LIN {X 0,Y 232.971,Z 461.148,A -85,B 0,C 180,E1 -19706.542,E2 -19706.542} C_VEL
LIN {X 0,Y 232.837,Z 461.984,A -85,B 0,C 180,E1 -19710.001,E2 -19710.001} C_VEL
LIN {X 0,Y 232.861,Z 461.79,A -85,B 0,C 180,E1 -19711.73,E2 -19711.73} C_VEL
LIN {X 0,Y 232.964,Z 461.204,A -85,B 0,C 180,E1 -19713.46,E2 -19713.46} C_VEL
LIN {X 0,Y 233.433,Z 458.881,A -85,B 0,C 180,E1 -19716.917,E2 -19716.917} C_VEL
LIN {X 0,Y 234.07,Z 456.015,A -85,B 0,C 180,E1 -19719.506,E2 -19719.506} C_VEL
LIN {X 0,Y 235.043,Z 452.127,A -85,B 0,C 180,E1 -19722.082,E2 -19722.082} C_VEL
LIN {X 0,Y 236.444,Z 447.107,A -85,B 0,C 180,E1 -19724.635,E2 -19724.635} C_VEL
LIN {X 0,Y 238.156,Z 440.785,A -85,B 0,C 180,E1 -19727.164,E2 -19727.164} C_VEL
LIN {X 0,Y 240.375,Z 432.868,A -85,B 0,C 180,E1 -19729.648,E2 -19729.648} C_VEL
LIN {X 0,Y 242.397,Z 424.824,A -85,B 0,C 180,E1 -19731.689,E2 -19731.689} C_VEL
LIN {X 0,Y 244.588,Z 414.953,A -85,B 0,C 180,E1 -19733.721,E2 -19733.721} C_VEL
LIN {X 0,Y 246.59,Z 405.255,A -85,B 0,C 180,E1 -19735.31,E2 -19735.31} C_VEL
LIN {X 0,Y 245.528,Z 395.502,A -85,B 0,C 180,E1 -19736.937,E2 -19736.937} C_VEL
LIN {X 0,Y 243.4,Z 384.419,A -85,B 0,C 180,E1 -19738.585,E2 -19738.585} C_VEL
LIN {X 0,Y 240.222,Z 372.784,A -85,B 0,C 180,E1 -19740.129,E2 -19740.129} C_VEL
LIN {X 0,Y 236.054,Z 361.103,A -85,B 0,C 180,E1 -19741.536,E2 -19741.536} C_VEL
LIN {X 0,Y 234.99,Z 358.228,A -85,B 0,C 180,E1 -19741.853,E2 -19741.853} C_VEL
LIN {X 0,Y 234.929,Z 357.743,A -85,B 0,C 180,E1 -19741.928,E2 -19741.928} C_VEL
LIN {X 0,Y 235.264,Z 354.456,A -85,B 0,C 180,E1 -19746.238,E2 -19746.238} C_VEL
LIN {X 0,Y 235.192,Z 352.491,A -85,B 0,C 180,E1 -19749.019,E2 -19749.019} C_VEL
LIN {X 0,Y 234.976,Z 350.772,A -85,B 0,C 180,E1 -19751.605,E2 -19751.605} C_VEL
LIN {X 0,Y 234.883,Z 350.23,A -85,B 0,C 180,E1 -19754.101,E2 -19754.101} C_VEL
LIN {X 0,Y 234.85,Z 350.231,A -85,B 0,C 180,E1 -19758.825,E2 -19758.825} C_VEL
LIN {X 0,Y 234.918,Z 350.222,A -85,B 0,C 180,E1 -19761.078,E2 -19761.078} C_VEL
LIN {X 0,Y 234.923,Z 350.221,A -85,B 0,C 180,E1 -19765.36,E2 -19765.36} C_VEL
LIN {X 0,Y 234.898,Z 350.226,A -85,B 0,C 180,E1 -19769.427,E2 -19769.427} C_VEL
LIN {X 0,Y 234.968,Z 350.214,A -85,B 0,C 180,E1 -19773.806,E2 -19773.806} C_VEL
LIN {X 0,Y 234.997,Z 350.214,A -85,B 0,C 180,E1 -19778.968,E2 -19778.968} C_VEL
LIN {X 0,Y 235.096,Z 350.201,A -85,B 0,C 180,E1 -19783.059,E2 -19783.059} C_VEL
LIN {X 0,Y 235.118,Z 350.195,A -85,B 0,C 180,E1 -19787.922,E2 -19787.922} C_VEL
LIN {X 0,Y 235.376,Z 350.164,A -85,B 0,C 180,E1 -19791.414,E2 -19791.414} C_VEL
LIN {X 0,Y 235.403,Z 350.16,A -85,B 0,C 180,E1 -19793.141,E2 -19793.141} C_VEL
LIN {X 0,Y 235.592,Z 350.139,A -85,B 0,C 180,E1 -19798.29,E2 -19798.29} C_VEL
LIN {X 0,Y 235.592,Z 350.137,A -85,B 0,C 180,E1 -19801.709,E2 -19801.709} C_VEL
LIN {X 0,Y 235.372,Z 350.166,A -85,B 0,C 180,E1 -19806.86,E2 -19806.86} C_VEL
LIN {X 0,Y 235.214,Z 350.187,A -85,B 0,C 180,E1 -19810.328,E2 -19810.328} C_VEL
LIN {X 0,Y 235.111,Z 350.201,A -85,B 0,C 180,E1 -19815.607,E2 -19815.607} C_VEL
LIN {X 0,Y 235.007,Z 350.213,A -85,B 0,C 180,E1 -19819.206,E2 -19819.206} C_VEL
LIN {X 0,Y 234.946,Z 350.219,A -85,B 0,C 180,E1 -19822.884,E2 -19822.884} C_VEL
LIN {X 0,Y 234.944,Z 350.219,A -85,B 0,C 180,E1 -19826.66,E2 -19826.66} C_VEL
LIN {X 0,Y 234.898,Z 350.227,A -85,B 0,C 180,E1 -19830.573,E2 -19830.573} C_VEL
LIN {X 0,Y 234.925,Z 350.225,A -85,B 0,C 180,E1 -19834.639,E2 -19834.639} C_VEL
LIN {X 0,Y 234.922,Z 350.234,A -85,B 0,C 180,E1 -19837.287,E2 -19837.287} C_VEL
LIN {X 0,Y 235.478,Z 353.686,A -85,B 0,C 180,E1 -19841.743,E2 -19841.743} C_VEL
LIN {X 0,Y 236.045,Z 356.925,A -85,B 0,C 180,E1 -19845.609,E2 -19845.609} C_VEL
LIN {X 0,Y 236.625,Z 360.143,A -85,B 0,C 180,E1 -19849.2,E2 -19849.2} C_VEL
LIN {X 0,Y 236.789,Z 361.71,A -85,B 0,C 180,E1 -19850.867,E2 -19850.867} C_VEL
LIN {X 0,Y 236.131,Z 362.697,A -85,B 0,C 180,E1 -19851.78,E2 -19851.78} C_VEL
LIN {X 0,Y 233.267,Z 364.499,A -85,B 0,C 180,E1 -19853.194,E2 -19853.194} C_VEL
LIN {X 0,Y 230.302,Z 366.325,A -85,B 0,C 180,E1 -19854.639,E2 -19854.639} C_VEL
LIN {X 0,Y 229.536,Z 367.356,A -85,B 0,C 180,E1 -19855.588,E2 -19855.588} C_VEL
LIN {X 0,Y 229.138,Z 369.003,A -85,B 0,C 180,E1 -19857.205,E2 -19857.205} C_VEL
LIN {X 0,Y 230.068,Z 372.388,A -85,B 0,C 180,E1 -19857.554,E2 -19857.554} C_VEL
LIN {X 0,Y 233.694,Z 385.256,A -85,B 0,C 180,E1 -19858.994,E2 -19858.994} C_VEL
LIN {X 0,Y 236.083,Z 397.637,A -85,B 0,C 180,E1 -19860.546,E2 -19860.546} C_VEL
LIN {X 0,Y 237.455,Z 409.332,A -85,B 0,C 180,E1 -19862.24,E2 -19862.24} C_VEL
LIN {X 0,Y 237.876,Z 420.833,A -85,B 0,C 180,E1 -19864.164,E2 -19864.164} C_VEL
LIN {X 0,Y 237.723,Z 425.768,A -85,B 0,C 180,E1 -19865.084,E2 -19865.084} C_VEL
LIN {X 0,Y 235.114,Z 436.231,A -85,B 0,C 180,E1 -19867.133,E2 -19867.133} C_VEL
LIN {X 0,Y 232.717,Z 445.972,A -85,B 0,C 180,E1 -19869.607,E2 -19869.607} C_VEL
LIN {X 0,Y 230.397,Z 454.218,A -85,B 0,C 180,E1 -19872.239,E2 -19872.239} C_VEL
LIN {X 0,Y 228.61,Z 460.648,A -85,B 0,C 180,E1 -19874.852,E2 -19874.852} C_VEL
LIN {X 0,Y 227.307,Z 465.76,A -85,B 0,C 180,E1 -19877.5,E2 -19877.5} C_VEL
LIN {X 0,Y 226.434,Z 469.734,A -85,B 0,C 180,E1 -19880.17,E2 -19880.17} C_VEL
LIN {X 0,Y 225.853,Z 472.672,A -85,B 0,C 180,E1 -19882.849,E2 -19882.849} C_VEL
LIN {X 0,Y 225.66,Z 474.484,A -85,B 0,C 180,E1 -19885.286,E2 -19885.286} C_VEL
LIN {X 0,Y 225.663,Z 475.686,A -85,B 0,C 180,E1 -19888.215,E2 -19888.215} C_VEL
LIN {X 0,Y 225.698,Z 475.901,A -85,B 0,C 180,E1 -19889.999,E2 -19889.999} C_VEL
LIN {X 0,Y 225.662,Z 475.678,A -85,B 0,C 180,E1 -19891.784,E2 -19891.784} C_VEL
LIN {X 0,Y 225.69,Z 474.056,A -85,B 0,C 180,E1 -19895.36,E2 -19895.36} C_VEL
LIN {X 0,Y 225.852,Z 472.648,A -85,B 0,C 180,E1 -19897.149,E2 -19897.149} C_VEL
LIN {X 0,Y 226.432,Z 469.698,A -85,B 0,C 180,E1 -19899.828,E2 -19899.828} C_VEL
LIN {X 0,Y 227.306,Z 465.709,A -85,B 0,C 180,E1 -19902.498,E2 -19902.498} C_VEL
LIN {X 0,Y 228.896,Z 459.582,A -85,B 0,C 180,E1 -19905.583,E2 -19905.583} C_VEL
LIN {X 0,Y 230.724,Z 452.894,A -85,B 0,C 180,E1 -19908.192,E2 -19908.192} C_VEL
LIN {X 0,Y 232.845,Z 444.953,A -85,B 0,C 180,E1 -19910.661,E2 -19910.661} C_VEL
LIN {X 0,Y 235.088,Z 436.095,A -85,B 0,C 180,E1 -19912.868,E2 -19912.868} C_VEL
LIN {X 0,Y 237.677,Z 425.596,A -85,B 0,C 180,E1 -19914.92,E2 -19914.92} C_VEL
LIN {X 0,Y 237.746,Z 415.806,A -85,B 0,C 180,E1 -19916.683,E2 -19916.683} C_VEL
LIN {X 0,Y 237.068,Z 405.419,A -85,B 0,C 180,E1 -19918.314,E2 -19918.314} C_VEL
LIN {X 0,Y 235.7,Z 395.253,A -85,B 0,C 180,E1 -19919.722,E2 -19919.722} C_VEL
LIN {X 0,Y 232.854,Z 382.031,A -85,B 0,C 180,E1 -19921.351,E2 -19921.351} C_VEL
LIN {X 0,Y 229.624,Z 371.42,A -85,B 0,C 180,E1 -19922.526,E2 -19922.526} C_VEL
LIN {X 0,Y 229.118,Z 368.985,A -85,B 0,C 180,E1 -19922.773,E2 -19922.773} C_VEL
LIN {X 0,Y 229.704,Z 366.183,A -85,B 0,C 180,E1 -19925.542,E2 -19925.542} C_VEL
LIN {X 0,Y 229.844,Z 363.042,A -85,B 0,C 180,E1 -19928.815,E2 -19928.815} C_VEL
LIN {X 0,Y 229.425,Z 359.571,A -85,B 0,C 180,E1 -19932.676,E2 -19932.676} C_VEL
LIN {X 0,Y 228.591,Z 355.533,A -85,B 0,C 180,E1 -19937.549,E2 -19937.549} C_VEL
LIN {X 0,Y 228.078,Z 352.174,A -85,B 0,C 180,E1 -19941.955,E2 -19941.955} C_VEL
LIN {X 0,Y 227.867,Z 351.102,A -85,B 0,C 180,E1 -19943.713,E2 -19943.713} C_VEL
LIN {X 0,Y 227.873,Z 351.102,A -85,B 0,C 180,E1 -19946.377,E2 -19946.377} C_VEL
LIN {X 0,Y 227.87,Z 351.104,A -85,B 0,C 180,E1 -19950.431,E2 -19950.431} C_VEL
LIN {X 0,Y 227.896,Z 351.099,A -85,B 0,C 180,E1 -19954.422,E2 -19954.422} C_VEL
LIN {X 0,Y 227.949,Z 351.091,A -85,B 0,C 180,E1 -19958.286,E2 -19958.286} C_VEL
LIN {X 0,Y 228.028,Z 351.081,A -85,B 0,C 180,E1 -19962.826,E2 -19962.826} C_VEL
LIN {X 0,Y 228.086,Z 351.073,A -85,B 0,C 180,E1 -19967.544,E2 -19967.544} C_VEL
LIN {X 0,Y 228.3,Z 351.046,A -85,B 0,C 180,E1 -19971.146,E2 -19971.146} C_VEL
LIN {X 0,Y 228.349,Z 351.04,A -85,B 0,C 180,E1 -19972.928,E2 -19972.928} C_VEL
LIN {X 0,Y 228.547,Z 351.016,A -85,B 0,C 180,E1 -19978.238,E2 -19978.238} C_VEL
LIN {X 0,Y 228.546,Z 351.016,A -85,B 0,C 180,E1 -19981.762,E2 -19981.762} C_VEL
LIN {X 0,Y 228.351,Z 351.041,A -85,B 0,C 180,E1 -19987.072,E2 -19987.072} C_VEL
LIN {X 0,Y 228.161,Z 351.063,A -85,B 0,C 180,E1 -19990.651,E2 -19990.651} C_VEL
LIN {X 0,Y 228.058,Z 351.074,A -85,B 0,C 180,E1 -19994.273,E2 -19994.273} C_VEL
LIN {X 0,Y 227.997,Z 351.084,A -85,B 0,C 180,E1 -19997.954,E2 -19997.954} C_VEL
LIN {X 0,Y 227.916,Z 351.092,A -85,B 0,C 180,E1 -20002.325,E2 -20002.325} C_VEL
LIN {X 0,Y 227.916,Z 351.095,A -85,B 0,C 180,E1 -20006.593,E2 -20006.593} C_VEL
LIN {X 0,Y 227.868,Z 351.101,A -85,B 0,C 180,E1 -20010.281,E2 -20010.281} C_VEL
LIN {X 0,Y 227.872,Z 351.1,A -85,B 0,C 180,E1 -20013.722,E2 -20013.722} C_VEL
LIN {X 0,Y 227.839,Z 351.104,A -85,B 0,C 180,E1 -20018.092,E2 -20018.092} C_VEL
LIN {X 0,Y 227.789,Z 351.111,A -85,B 0,C 180,E1 -20022.748,E2 -20022.748} C_VEL
LIN {X 0,Y 227.855,Z 351.213,A -85,B 0,C 180,E1 -20027.27,E2 -20027.27} C_VEL
LIN {X 0,Y 228.109,Z 353.189,A -85,B 0,C 180,E1 -20030.376,E2 -20030.376} C_VEL
LIN {X 0,Y 228.239,Z 355.821,A -85,B 0,C 180,E1 -20034.195,E2 -20034.195} C_VEL
LIN {X 0,Y 228.018,Z 357.999,A -85,B 0,C 180,E1 -20037.156,E2 -20037.156} C_VEL
LIN {X 0,Y 229.088,Z 361.247,A -85,B 0,C 180,E1 -20037.526,E2 -20037.526} C_VEL
LIN {X 0,Y 233.181,Z 372.217,A -85,B 0,C 180,E1 -20038.935,E2 -20038.935} C_VEL
LIN {X 0,Y 236.434,Z 383.735,A -85,B 0,C 180,E1 -20040.529,E2 -20040.529} C_VEL
LIN {X 0,Y 238.509,Z 394.227,A -85,B 0,C 180,E1 -20042.128,E2 -20042.128} C_VEL
LIN {X 0,Y 239.672,Z 403.1,A -85,B 0,C 180,E1 -20043.639,E2 -20043.639} C_VEL
LIN {X 0,Y 239.797,Z 407.32,A -85,B 0,C 180,E1 -20044.388,E2 -20044.388} C_VEL
LIN {X 0,Y 237.437,Z 417.763,A -85,B 0,C 180,E1 -20046.218,E2 -20046.218} C_VEL
LIN {X 0,Y 235.421,Z 426.646,A -85,B 0,C 180,E1 -20048.185,E2 -20048.185} C_VEL
LIN {X 0,Y 232.983,Z 435.524,A -85,B 0,C 180,E1 -20050.622,E2 -20050.622} C_VEL
LIN {X 0,Y 230.792,Z 442.926,A -85,B 0,C 180,E1 -20053.186,E2 -20053.186} C_VEL
LIN {X 0,Y 229.094,Z 448.862,A -85,B 0,C 180,E1 -20055.794,E2 -20055.794} C_VEL
LIN {X 0,Y 227.744,Z 453.551,A -85,B 0,C 180,E1 -20058.43,E2 -20058.43} C_VEL
LIN {X 0,Y 226.795,Z 457.137,A -85,B 0,C 180,E1 -20061.088,E2 -20061.088} C_VEL
LIN {X 0,Y 226.238,Z 459.716,A -85,B 0,C 180,E1 -20063.76,E2 -20063.76} C_VEL
LIN {X 0,Y 225.881,Z 461.364,A -85,B 0,C 180,E1 -20066.433,E2 -20066.433} C_VEL
LIN {X 0,Y 225.778,Z 461.971,A -85,B 0,C 180,E1 -20068.217,E2 -20068.217} C_VEL
LIN {X 0,Y 225.751,Z 462.199,A -85,B 0,C 180,E1 -20070.001,E2 -20070.001} C_VEL
LIN {X 0,Y 225.778,Z 462.005,A -85,B 0,C 180,E1 -20071.785,E2 -20071.785} C_VEL
LIN {X 0,Y 226.06,Z 460.453,A -85,B 0,C 180,E1 -20075.352,E2 -20075.352} C_VEL
LIN {X 0,Y 226.394,Z 459.096,A -85,B 0,C 180,E1 -20077.134,E2 -20077.134} C_VEL
LIN {X 0,Y 227.07,Z 456.23,A -85,B 0,C 180,E1 -20079.802,E2 -20079.802} C_VEL
LIN {X 0,Y 228.109,Z 452.341,A -85,B 0,C 180,E1 -20082.455,E2 -20082.455} C_VEL
LIN {X 0,Y 229.581,Z 447.321,A -85,B 0,C 180,E1 -20085.083,E2 -20085.083} C_VEL
LIN {X 0,Y 231.38,Z 440.998,A -85,B 0,C 180,E1 -20087.683,E2 -20087.683} C_VEL
LIN {X 0,Y 233.706,Z 433.08,A -85,B 0,C 180,E1 -20090.233,E2 -20090.233} C_VEL
LIN {X 0,Y 235.703,Z 425.511,A -85,B 0,C 180,E1 -20092.214,E2 -20092.214} C_VEL
LIN {X 0,Y 237.845,Z 416.231,A -85,B 0,C 180,E1 -20094.204,E2 -20094.204} C_VEL
LIN {X 0,Y 239.95,Z 406.756,A -85,B 0,C 180,E1 -20095.829,E2 -20095.829} C_VEL
LIN {X 0,Y 239.062,Z 397.402,A -85,B 0,C 180,E1 -20097.473,E2 -20097.473} C_VEL
LIN {X 0,Y 237.101,Z 386.551,A -85,B 0,C 180,E1 -20099.192,E2 -20099.192} C_VEL
LIN {X 0,Y 234.225,Z 375.555,A -85,B 0,C 180,E1 -20100.763,E2 -20100.763} C_VEL
LIN {X 0,Y 230.277,Z 364.192,A -85,B 0,C 180,E1 -20102.255,E2 -20102.255} C_VEL
LIN {X 0,Y 228.124,Z 358.66,A -85,B 0,C 180,E1 -20102.921,E2 -20102.921} C_VEL
LIN {X 0,Y 228.02,Z 357.983,A -85,B 0,C 180,E1 -20103.015,E2 -20103.015} C_VEL
LIN {X 0,Y 228.248,Z 355.211,A -85,B 0,C 180,E1 -20106.815,E2 -20106.815} C_VEL
LIN {X 0,Y 228.052,Z 352.842,A -85,B 0,C 180,E1 -20110.329,E2 -20110.329} C_VEL
LIN {X 0,Y 227.856,Z 351.327,A -85,B 0,C 180,E1 -20112.732,E2 -20112.732} C_VEL
LIN {X 0,Y 227.821,Z 351.11,A -85,B 0,C 180,E1 -20115.196,E2 -20115.196} C_VEL
LIN {X 0,Y 227.798,Z 351.111,A -85,B 0,C 180,E1 -20119.617,E2 -20119.617} C_VEL
LIN {X 0,Y 227.864,Z 351.101,A -85,B 0,C 180,E1 -20124.125,E2 -20124.125} C_VEL
LIN {X 0,Y 227.856,Z 351.099,A -85,B 0,C 180,E1 -20128.375,E2 -20128.375} C_VEL
LIN {X 0,Y 227.854,Z 351.101,A -85,B 0,C 180,E1 -20132.441,E2 -20132.441} C_VEL
LIN {X 0,Y 227.894,Z 351.096,A -85,B 0,C 180,E1 -20136.365,E2 -20136.365} C_VEL
LIN {X 0,Y 227.937,Z 351.091,A -85,B 0,C 180,E1 -20140.174,E2 -20140.174} C_VEL
LIN {X 0,Y 228.057,Z 351.076,A -85,B 0,C 180,E1 -20143.898,E2 -20143.898} C_VEL
LIN {X 0,Y 228.074,Z 351.073,A -85,B 0,C 180,E1 -20147.543,E2 -20147.543} C_VEL
LIN {X 0,Y 228.306,Z 351.046,A -85,B 0,C 180,E1 -20151.146,E2 -20151.146} C_VEL
LIN {X 0,Y 228.354,Z 351.039,A -85,B 0,C 180,E1 -20152.928,E2 -20152.928} C_VEL
LIN {X 0,Y 228.551,Z 351.016,A -85,B 0,C 180,E1 -20158.238,E2 -20158.238} C_VEL
LIN {X 0,Y 228.551,Z 351.014,A -85,B 0,C 180,E1 -20161.762,E2 -20161.762} C_VEL
LIN {X 0,Y 228.323,Z 351.044,A -85,B 0,C 180,E1 -20167.072,E2 -20167.072} C_VEL
LIN {X 0,Y 228.145,Z 351.066,A -85,B 0,C 180,E1 -20170.651,E2 -20170.651} C_VEL
LIN {X 0,Y 228.062,Z 351.08,A -85,B 0,C 180,E1 -20174.272,E2 -20174.272} C_VEL
LIN {X 0,Y 228.002,Z 351.086,A -85,B 0,C 180,E1 -20177.953,E2 -20177.953} C_VEL
LIN {X 0,Y 227.921,Z 351.094,A -85,B 0,C 180,E1 -20182.324,E2 -20182.324} C_VEL
LIN {X 0,Y 227.922,Z 351.094,A -85,B 0,C 180,E1 -20186.592,E2 -20186.592} C_VEL
LIN {X 0,Y 227.873,Z 351.102,A -85,B 0,C 180,E1 -20190.281,E2 -20190.281} C_VEL
LIN {X 0,Y 227.876,Z 351.103,A -85,B 0,C 180,E1 -20193.721,E2 -20193.721} C_VEL
LIN {X 0,Y 227.916,Z 351.27,A -85,B 0,C 180,E1 -20196.704,E2 -20196.704} C_VEL
LIN {X 0,Y 228.32,Z 353.894,A -85,B 0,C 180,E1 -20200.272,E2 -20200.272} C_VEL
LIN {X 0,Y 228.979,Z 357.739,A -85,B 0,C 180,E1 -20205.095,E2 -20205.095} C_VEL
LIN {X 0,Y 229.569,Z 360.957,A -85,B 0,C 180,E1 -20208.839,E2 -20208.839} C_VEL
LIN {X 0,Y 229.799,Z 364.142,A -85,B 0,C 180,E1 -20212.29,E2 -20212.29} C_VEL
LIN {X 0,Y 229.536,Z 367.356,A -85,B 0,C 180,E1 -20215.588,E2 -20215.588} C_VEL
LIN {X 0,Y 229.594,Z 369.045,A -85,B 0,C 180,E1 -20216.42,E2 -20216.42} C_VEL
LIN {X 0,Y 229.811,Z 371.78,A -85,B 0,C 180,E1 -20217.075,E2 -20217.075} C_VEL
LIN {X 0,Y 230.043,Z 376.979,A -85,B 0,C 180,E1 -20217.779,E2 -20217.779} C_VEL
LIN {X 0,Y 229.617,Z 387.244,A -85,B 0,C 180,E1 -20218.563,E2 -20218.563} C_VEL
LIN {X 0,Y 228.964,Z 393.373,A -85,B 0,C 180,E1 -20219.082,E2 -20219.082} C_VEL
LIN {X 0,Y 229.078,Z 395.306,A -85,B 0,C 180,E1 -20219.316,E2 -20219.316} C_VEL
LIN {X 0,Y 230.658,Z 407.037,A -85,B 0,C 180,E1 -20221.043,E2 -20221.043} C_VEL
LIN {X 0,Y 231.246,Z 417.991,A -85,B 0,C 180,E1 -20222.878,E2 -20222.878} C_VEL
LIN {X 0,Y 230.995,Z 426.732,A -85,B 0,C 180,E1 -20224.548,E2 -20224.548} C_VEL
LIN {X 0,Y 228.568,Z 436.018,A -85,B 0,C 180,E1 -20226.439,E2 -20226.439} C_VEL
LIN {X 0,Y 226.272,Z 444.877,A -85,B 0,C 180,E1 -20228.717,E2 -20228.717} C_VEL
LIN {X 0,Y 223.961,Z 452.766,A -85,B 0,C 180,E1 -20231.237,E2 -20231.237} C_VEL
LIN {X 0,Y 222.045,Z 459.438,A -85,B 0,C 180,E1 -20233.921,E2 -20233.921} C_VEL
LIN {X 0,Y 220.35,Z 465.545,A -85,B 0,C 180,E1 -20237.099,E2 -20237.099} C_VEL
LIN {X 0,Y 219.406,Z 469.519,A -85,B 0,C 180,E1 -20239.852,E2 -20239.852} C_VEL
LIN {X 0,Y 218.804,Z 472.457,A -85,B 0,C 180,E1 -20242.618,E2 -20242.618} C_VEL
LIN {X 0,Y 218.576,Z 474.428,A -85,B 0,C 180,E1 -20245.39,E2 -20245.39} C_VEL
LIN {X 0,Y 218.56,Z 475.47,A -85,B 0,C 180,E1 -20248.157,E2 -20248.157} C_VEL
LIN {X 0,Y 218.614,Z 475.686,A -85,B 0,C 180,E1 -20249.999,E2 -20249.999} C_VEL
LIN {X 0,Y 218.56,Z 475.462,A -85,B 0,C 180,E1 -20251.842,E2 -20251.842} C_VEL
LIN {X 0,Y 218.554,Z 474.453,A -85,B 0,C 180,E1 -20254.538,E2 -20254.538} C_VEL
LIN {X 0,Y 218.802,Z 472.432,A -85,B 0,C 180,E1 -20257.381,E2 -20257.381} C_VEL
LIN {X 0,Y 219.404,Z 469.481,A -85,B 0,C 180,E1 -20260.146,E2 -20260.146} C_VEL
LIN {X 0,Y 220.349,Z 465.491,A -85,B 0,C 180,E1 -20262.9,E2 -20262.9} C_VEL
LIN {X 0,Y 222.044,Z 459.364,A -85,B 0,C 180,E1 -20266.077,E2 -20266.077} C_VEL
LIN {X 0,Y 223.965,Z 452.675,A -85,B 0,C 180,E1 -20268.761,E2 -20268.761} C_VEL
LIN {X 0,Y 225.998,Z 445.402,A -85,B 0,C 180,E1 -20271.103,E2 -20271.103} C_VEL
LIN {X 0,Y 228.541,Z 435.876,A -85,B 0,C 180,E1 -20273.562,E2 -20273.562} C_VEL
LIN {X 0,Y 231.097,Z 425.371,A -85,B 0,C 180,E1 -20275.68,E2 -20275.68} C_VEL
LIN {X 0,Y 231.068,Z 414.45,A -85,B 0,C 180,E1 -20277.71,E2 -20277.71} C_VEL
LIN {X 0,Y 230.276,Z 403.806,A -85,B 0,C 180,E1 -20279.422,E2 -20279.422} C_VEL
LIN {X 0,Y 228.576,Z 392.654,A -85,B 0,C 180,E1 -20281.011,E2 -20281.011} C_VEL
LIN {X 0,Y 225.776,Z 380.579,A -85,B 0,C 180,E1 -20282.543,E2 -20282.543} C_VEL
LIN {X 0,Y 222.419,Z 369.35,A -85,B 0,C 180,E1 -20283.814,E2 -20283.814} C_VEL
LIN {X 0,Y 222.35,Z 368.792,A -85,B 0,C 180,E1 -20283.861,E2 -20283.861} C_VEL
LIN {X 0,Y 222.795,Z 364.916,A -85,B 0,C 180,E1 -20287.943,E2 -20287.943} C_VEL
LIN {X 0,Y 222.639,Z 362.413,A -85,B 0,C 180,E1 -20290.746,E2 -20290.746} C_VEL
LIN {X 0,Y 222.147,Z 359.583,A -85,B 0,C 180,E1 -20294.105,E2 -20294.105} C_VEL
LIN {X 0,Y 221.52,Z 356.342,A -85,B 0,C 180,E1 -20298.221,E2 -20298.221} C_VEL
LIN {X 0,Y 220.992,Z 352.997,A -85,B 0,C 180,E1 -20302.826,E2 -20302.826} C_VEL
LIN {X 0,Y 220.817,Z 351.98,A -85,B 0,C 180,E1 -20304.49,E2 -20304.49} C_VEL
LIN {X 0,Y 220.829,Z 351.979,A -85,B 0,C 180,E1 -20309.389,E2 -20309.389} C_VEL
LIN {X 0,Y 220.869,Z 351.974,A -85,B 0,C 180,E1 -20313.546,E2 -20313.546} C_VEL
LIN {X 0,Y 220.862,Z 351.974,A -85,B 0,C 180,E1 -20317.552,E2 -20317.552} C_VEL
LIN {X 0,Y 220.978,Z 351.96,A -85,B 0,C 180,E1 -20322.571,E2 -20322.571} C_VEL
LIN {X 0,Y 221.018,Z 351.953,A -85,B 0,C 180,E1 -20327.139,E2 -20327.139} C_VEL
LIN {X 0,Y 221.23,Z 351.927,A -85,B 0,C 180,E1 -20330.861,E2 -20330.861} C_VEL
LIN {X 0,Y 221.284,Z 351.92,A -85,B 0,C 180,E1 -20332.701,E2 -20332.701} C_VEL
LIN {X 0,Y 221.505,Z 351.893,A -85,B 0,C 180,E1 -20338.182,E2 -20338.182} C_VEL
LIN {X 0,Y 221.504,Z 351.893,A -85,B 0,C 180,E1 -20341.818,E2 -20341.818} C_VEL
LIN {X 0,Y 221.304,Z 351.92,A -85,B 0,C 180,E1 -20347.298,E2 -20347.298} C_VEL
LIN {X 0,Y 221.105,Z 351.943,A -85,B 0,C 180,E1 -20350.995,E2 -20350.995} C_VEL
LIN {X 0,Y 221.01,Z 351.954,A -85,B 0,C 180,E1 -20356.63,E2 -20356.63} C_VEL
LIN {X 0,Y 220.881,Z 351.97,A -85,B 0,C 180,E1 -20360.487,E2 -20360.487} C_VEL
LIN {X 0,Y 220.842,Z 351.975,A -85,B 0,C 180,E1 -20364.438,E2 -20364.438} C_VEL
LIN {X 0,Y 220.798,Z 351.982,A -85,B 0,C 180,E1 -20368.519,E2 -20368.519} C_VEL
LIN {X 0,Y 220.807,Z 351.981,A -85,B 0,C 180,E1 -20372.758,E2 -20372.758} C_VEL
LIN {X 0,Y 220.805,Z 351.98,A -85,B 0,C 180,E1 -20377.279,E2 -20377.279} C_VEL
LIN {X 0,Y 220.748,Z 351.987,A -85,B 0,C 180,E1 -20381.958,E2 -20381.958} C_VEL
LIN {X 0,Y 220.773,Z 351.984,A -85,B 0,C 180,E1 -20385.548,E2 -20385.548} C_VEL
LIN {X 0,Y 220.841,Z 352.362,A -85,B 0,C 180,E1 -20387.05,E2 -20387.05} C_VEL
LIN {X 0,Y 221.124,Z 354.511,A -85,B 0,C 180,E1 -20390.533,E2 -20390.533} C_VEL
LIN {X 0,Y 221.222,Z 356.062,A -85,B 0,C 180,E1 -20392.873,E2 -20392.873} C_VEL
LIN {X 0,Y 221.068,Z 358.265,A -85,B 0,C 180,E1 -20396.004,E2 -20396.004} C_VEL
LIN {X 0,Y 222.308,Z 361.658,A -85,B 0,C 180,E1 -20396.416,E2 -20396.416} C_VEL
LIN {X 0,Y 226.747,Z 373.513,A -85,B 0,C 180,E1 -20398.042,E2 -20398.042} C_VEL
LIN {X 0,Y 230.038,Z 385.159,A -85,B 0,C 180,E1 -20399.759,E2 -20399.759} C_VEL
LIN {X 0,Y 232.035,Z 395.634,A -85,B 0,C 180,E1 -20401.447,E2 -20401.447} C_VEL
LIN {X 0,Y 233.178,Z 404.943,A -85,B 0,C 180,E1 -20403.123,E2 -20403.123} C_VEL
LIN {X 0,Y 233.346,Z 407.542,A -85,B 0,C 180,E1 -20403.626,E2 -20403.626} C_VEL
LIN {X 0,Y 230.948,Z 417.983,A -85,B 0,C 180,E1 -20405.506,E2 -20405.506} C_VEL
LIN {X 0,Y 228.76,Z 427.167,A -85,B 0,C 180,E1 -20407.598,E2 -20407.598} C_VEL
LIN {X 0,Y 226.305,Z 435.742,A -85,B 0,C 180,E1 -20410.026,E2 -20410.026} C_VEL
LIN {X 0,Y 224,Z 443.144,A -85,B 0,C 180,E1 -20412.66,E2 -20412.66} C_VEL
LIN {X 0,Y 222.212,Z 449.079,A -85,B 0,C 180,E1 -20415.345,E2 -20415.345} C_VEL
LIN {X 0,Y 220.798,Z 453.768,A -85,B 0,C 180,E1 -20418.061,E2 -20418.061} C_VEL
LIN {X 0,Y 219.788,Z 457.353,A -85,B 0,C 180,E1 -20420.801,E2 -20420.801} C_VEL
LIN {X 0,Y 219.119,Z 460.183,A -85,B 0,C 180,E1 -20423.878,E2 -20423.878} C_VEL
LIN {X 0,Y 218.793,Z 461.58,A -85,B 0,C 180,E1 -20426.317,E2 -20426.317} C_VEL
LIN {X 0,Y 218.697,Z 462.187,A -85,B 0,C 180,E1 -20428.159,E2 -20428.159} C_VEL
LIN {X 0,Y 218.666,Z 462.414,A -85,B 0,C 180,E1 -20430.001,E2 -20430.001} C_VEL
LIN {X 0,Y 218.696,Z 462.22,A -85,B 0,C 180,E1 -20431.842,E2 -20431.842} C_VEL
LIN {X 0,Y 218.995,Z 460.668,A -85,B 0,C 180,E1 -20435.525,E2 -20435.525} C_VEL
LIN {X 0,Y 219.352,Z 459.31,A -85,B 0,C 180,E1 -20437.364,E2 -20437.364} C_VEL
LIN {X 0,Y 220.072,Z 456.445,A -85,B 0,C 180,E1 -20440.117,E2 -20440.117} C_VEL
LIN {X 0,Y 221.189,Z 452.555,A -85,B 0,C 180,E1 -20442.852,E2 -20442.852} C_VEL
LIN {X 0,Y 222.734,Z 447.535,A -85,B 0,C 180,E1 -20445.558,E2 -20445.558} C_VEL
LIN {X 0,Y 224.631,Z 441.211,A -85,B 0,C 180,E1 -20448.233,E2 -20448.233} C_VEL
LIN {X 0,Y 227.066,Z 433.293,A -85,B 0,C 180,E1 -20450.852,E2 -20450.852} C_VEL
LIN {X 0,Y 229.022,Z 426.217,A -85,B 0,C 180,E1 -20452.766,E2 -20452.766} C_VEL
LIN {X 0,Y 231.378,Z 416.443,A -85,B 0,C 180,E1 -20454.926,E2 -20454.926} C_VEL
LIN {X 0,Y 233.327,Z 408.253,A -85,B 0,C 180,E1 -20456.378,E2 -20456.378} C_VEL
LIN {X 0,Y 232.672,Z 399.6,A -85,B 0,C 180,E1 -20457.984,E2 -20457.984} C_VEL
LIN {X 0,Y 230.862,Z 388.892,A -85,B 0,C 180,E1 -20459.789,E2 -20459.789} C_VEL
LIN {X 0,Y 228.071,Z 377.711,A -85,B 0,C 180,E1 -20461.493,E2 -20461.493} C_VEL
LIN {X 0,Y 224.198,Z 366.379,A -85,B 0,C 180,E1 -20463.096,E2 -20463.096} C_VEL
LIN {X 0,Y 221.94,Z 361.042,A -85,B 0,C 180,E1 -20463.832,E2 -20463.832} C_VEL
LIN {X 0,Y 221.062,Z 358.241,A -85,B 0,C 180,E1 -20464.187,E2 -20464.187} C_VEL
LIN {X 0,Y 221.222,Z 355.972,A -85,B 0,C 180,E1 -20467.418,E2 -20467.418} C_VEL
LIN {X 0,Y 221.082,Z 354.102,A -85,B 0,C 180,E1 -20470.276,E2 -20470.276} C_VEL
LIN {X 0,Y 220.843,Z 352.469,A -85,B 0,C 180,E1 -20472.95,E2 -20472.95} C_VEL
LIN {X 0,Y 220.772,Z 351.989,A -85,B 0,C 180,E1 -20474.455,E2 -20474.455} C_VEL
LIN {X 0,Y 220.749,Z 351.989,A -85,B 0,C 180,E1 -20478.042,E2 -20478.042} C_VEL
LIN {X 0,Y 220.825,Z 351.977,A -85,B 0,C 180,E1 -20482.793,E2 -20482.793} C_VEL
LIN {X 0,Y 220.812,Z 351.979,A -85,B 0,C 180,E1 -20487.243,E2 -20487.243} C_VEL
LIN {X 0,Y 220.803,Z 351.978,A -85,B 0,C 180,E1 -20491.482,E2 -20491.482} C_VEL
LIN {X 0,Y 220.847,Z 351.973,A -85,B 0,C 180,E1 -20495.562,E2 -20495.562} C_VEL
LIN {X 0,Y 220.887,Z 351.97,A -85,B 0,C 180,E1 -20499.513,E2 -20499.513} C_VEL
LIN {X 0,Y 221.016,Z 351.954,A -85,B 0,C 180,E1 -20503.37,E2 -20503.37} C_VEL
LIN {X 0,Y 221.106,Z 351.944,A -85,B 0,C 180,E1 -20509.005,E2 -20509.005} C_VEL
LIN {X 0,Y 221.289,Z 351.92,A -85,B 0,C 180,E1 -20512.701,E2 -20512.701} C_VEL
LIN {X 0,Y 221.51,Z 351.893,A -85,B 0,C 180,E1 -20518.182,E2 -20518.182} C_VEL
LIN {X 0,Y 221.509,Z 351.892,A -85,B 0,C 180,E1 -20521.818,E2 -20521.818} C_VEL
LIN {X 0,Y 221.258,Z 351.925,A -85,B 0,C 180,E1 -20527.299,E2 -20527.299} C_VEL
LIN {X 0,Y 221.067,Z 351.948,A -85,B 0,C 180,E1 -20530.996,E2 -20530.996} C_VEL
LIN {X 0,Y 221.016,Z 351.956,A -85,B 0,C 180,E1 -20536.63,E2 -20536.63} C_VEL
LIN {X 0,Y 220.887,Z 351.971,A -85,B 0,C 180,E1 -20540.487,E2 -20540.487} C_VEL
LIN {X 0,Y 220.847,Z 351.975,A -85,B 0,C 180,E1 -20544.437,E2 -20544.437} C_VEL
LIN {X 0,Y 220.803,Z 351.982,A -85,B 0,C 180,E1 -20548.518,E2 -20548.518} C_VEL
LIN {X 0,Y 220.812,Z 351.983,A -85,B 0,C 180,E1 -20552.757,E2 -20552.757} C_VEL
LIN {X 0,Y 220.846,Z 352.105,A -85,B 0,C 180,E1 -20555.785,E2 -20555.785} C_VEL
LIN {X 0,Y 221.376,Z 355.332,A -85,B 0,C 180,E1 -20560.366,E2 -20560.366} C_VEL
LIN {X 0,Y 221.811,Z 358.294,A -85,B 0,C 180,E1 -20564.192,E2 -20564.192} C_VEL
LIN {X 0,Y 222.514,Z 361.769,A -85,B 0,C 180,E1 -20568.45,E2 -20568.45} C_VEL
LIN {X 0,Y 222.769,Z 364.981,A -85,B 0,C 180,E1 -20572.065,E2 -20572.065} C_VEL
LIN {X 0,Y 222.371,Z 368.77,A -85,B 0,C 180,E1 -20576.059,E2 -20576.059} C_VEL
LIN {X 0,Y 224.417,Z 375.692,A -85,B 0,C 180,E1 -20576.838,E2 -20576.838} C_VEL
LIN {X 0,Y 227.691,Z 388.021,A -85,B 0,C 180,E1 -20578.35,E2 -20578.35} C_VEL
LIN {X 0,Y 229.078,Z 395.306,A -85,B 0,C 180,E1 -20579.316,E2 -20579.316} C_VEL
LIN {X 0,Y 229.32,Z 398.835,A -85,B 0,C 180,E1 -20579.764,E2 -20579.764} C_VEL
LIN {X 0,Y 228.367,Z 405.997,A -85,B 0,C 180,E1 -20580.58,E2 -20580.58} C_VEL
LIN {X 0,Y 225.215,Z 418.131,A -85,B 0,C 180,E1 -20582.138,E2 -20582.138} C_VEL
LIN {X 0,Y 224.603,Z 422.96,A -85,B 0,C 180,E1 -20583.017,E2 -20583.017} C_VEL
LIN {X 0,Y 224.295,Z 427.648,A -85,B 0,C 180,E1 -20583.98,E2 -20583.98} C_VEL
LIN {X 0,Y 221.536,Z 437.6,A -85,B 0,C 180,E1 -20586.141,E2 -20586.141} C_VEL
LIN {X 0,Y 219.034,Z 446.848,A -85,B 0,C 180,E1 -20588.702,E2 -20588.702} C_VEL
LIN {X 0,Y 216.491,Z 454.947,A -85,B 0,C 180,E1 -20591.547,E2 -20591.547} C_VEL
LIN {X 0,Y 214.289,Z 462.04,A -85,B 0,C 180,E1 -20594.788,E2 -20594.788} C_VEL
LIN {X 0,Y 213.01,Z 466.765,A -85,B 0,C 180,E1 -20597.616,E2 -20597.616} C_VEL
LIN {X 0,Y 212.134,Z 470.378,A -85,B 0,C 180,E1 -20600.464,E2 -20600.464} C_VEL
LIN {X 0,Y 211.735,Z 472.241,A -85,B 0,C 180,E1 -20602.37,E2 -20602.37} C_VEL
LIN {X 0,Y 211.474,Z 474.377,A -85,B 0,C 180,E1 -20605.565,E2 -20605.565} C_VEL
LIN {X 0,Y 211.461,Z 475.255,A -85,B 0,C 180,E1 -20608.095,E2 -20608.095} C_VEL
LIN {X 0,Y 211.532,Z 475.471,A -85,B 0,C 180,E1 -20609.999,E2 -20609.999} C_VEL
LIN {X 0,Y 211.46,Z 475.246,A -85,B 0,C 180,E1 -20611.904,E2 -20611.904} C_VEL
LIN {X 0,Y 211.473,Z 474.365,A -85,B 0,C 180,E1 -20614.433,E2 -20614.433} C_VEL
LIN {X 0,Y 211.733,Z 472.215,A -85,B 0,C 180,E1 -20617.629,E2 -20617.629} C_VEL
LIN {X 0,Y 212.398,Z 469.264,A -85,B 0,C 180,E1 -20620.485,E2 -20620.485} C_VEL
LIN {X 0,Y 213.38,Z 465.273,A -85,B 0,C 180,E1 -20623.329,E2 -20623.329} C_VEL
LIN {X 0,Y 215.185,Z 459.145,A -85,B 0,C 180,E1 -20626.604,E2 -20626.604} C_VEL
LIN {X 0,Y 217.241,Z 452.458,A -85,B 0,C 180,E1 -20629.365,E2 -20629.365} C_VEL
LIN {X 0,Y 219.617,Z 444.261,A -85,B 0,C 180,E1 -20632.052,E2 -20632.052} C_VEL
LIN {X 0,Y 222.021,Z 435.657,A -85,B 0,C 180,E1 -20634.298,E2 -20634.298} C_VEL
LIN {X 0,Y 224.423,Z 426.328,A -85,B 0,C 180,E1 -20636.252,E2 -20636.252} C_VEL
LIN {X 0,Y 224.548,Z 416.569,A -85,B 0,C 180,E1 -20638.172,E2 -20638.172} C_VEL
LIN {X 0,Y 223.828,Z 404.947,A -85,B 0,C 180,E1 -20640.156,E2 -20640.156} C_VEL
LIN {X 0,Y 222.008,Z 392.705,A -85,B 0,C 180,E1 -20642.001,E2 -20642.001} C_VEL
LIN {X 0,Y 219.243,Z 380.81,A -85,B 0,C 180,E1 -20643.603,E2 -20643.603} C_VEL
LIN {X 0,Y 215.568,Z 368.901,A -85,B 0,C 180,E1 -20645.051,E2 -20645.051} C_VEL
LIN {X 0,Y 215.529,Z 368.424,A -85,B 0,C 180,E1 -20645.227,E2 -20645.227} C_VEL
LIN {X 0,Y 215.8,Z 365.385,A -85,B 0,C 180,E1 -20648.591,E2 -20648.591} C_VEL
LIN {X 0,Y 215.564,Z 362.982,A -85,B 0,C 180,E1 -20651.421,E2 -20651.421} C_VEL
LIN {X 0,Y 214.852,Z 359.324,A -85,B 0,C 180,E1 -20656.022,E2 -20656.022} C_VEL
LIN {X 0,Y 214.466,Z 357.068,A -85,B 0,C 180,E1 -20659.05,E2 -20659.05} C_VEL
LIN {X 0,Y 213.95,Z 353.809,A -85,B 0,C 180,E1 -20663.752,E2 -20663.752} C_VEL
LIN {X 0,Y 213.761,Z 352.859,A -85,B 0,C 180,E1 -20665.277,E2 -20665.277} C_VEL
LIN {X 0,Y 213.763,Z 352.861,A -85,B 0,C 180,E1 -20668.736,E2 -20668.736} C_VEL
LIN {X 0,Y 213.782,Z 352.857,A -85,B 0,C 180,E1 -20672.597,E2 -20672.597} C_VEL
LIN {X 0,Y 213.805,Z 352.853,A -85,B 0,C 180,E1 -20676.978,E2 -20676.978} C_VEL
LIN {X 0,Y 213.937,Z 352.836,A -85,B 0,C 180,E1 -20682.803,E2 -20682.803} C_VEL
LIN {X 0,Y 213.973,Z 352.831,A -85,B 0,C 180,E1 -20686.708,E2 -20686.708} C_VEL
LIN {X 0,Y 214.161,Z 352.808,A -85,B 0,C 180,E1 -20690.556,E2 -20690.556} C_VEL
LIN {X 0,Y 214.222,Z 352.801,A -85,B 0,C 180,E1 -20692.459,E2 -20692.459} C_VEL
LIN {X 0,Y 214.439,Z 352.774,A -85,B 0,C 180,E1 -20698.122,E2 -20698.122} C_VEL
LIN {X 0,Y 214.528,Z 352.762,A -85,B 0,C 180,E1 -20700,E2 -20700} C_VEL
LIN {X 0,Y 214.438,Z 352.772,A -85,B 0,C 180,E1 -20701.878,E2 -20701.878} C_VEL
LIN {X 0,Y 214.241,Z 352.798,A -85,B 0,C 180,E1 -20707.54,E2 -20707.54} C_VEL
LIN {X 0,Y 214.02,Z 352.825,A -85,B 0,C 180,E1 -20711.363,E2 -20711.363} C_VEL
LIN {X 0,Y 213.928,Z 352.838,A -85,B 0,C 180,E1 -20715.237,E2 -20715.237} C_VEL
LIN {X 0,Y 213.831,Z 352.849,A -85,B 0,C 180,E1 -20719.188,E2 -20719.188} C_VEL
LIN {X 0,Y 213.797,Z 352.855,A -85,B 0,C 180,E1 -20723.233,E2 -20723.233} C_VEL
LIN {X 0,Y 213.781,Z 352.856,A -85,B 0,C 180,E1 -20727.429,E2 -20727.429} C_VEL
LIN {X 0,Y 213.754,Z 352.859,A -85,B 0,C 180,E1 -20731.74,E2 -20731.74} C_VEL
LIN {X 0,Y 213.739,Z 352.861,A -85,B 0,C 180,E1 -20736.289,E2 -20736.289} C_VEL
LIN {X 0,Y 213.695,Z 352.864,A -85,B 0,C 180,E1 -20741.13,E2 -20741.13} C_VEL
LIN {X 0,Y 213.699,Z 352.864,A -85,B 0,C 180,E1 -20743.681,E2 -20743.681} C_VEL
LIN {X 0,Y 213.774,Z 353.24,A -85,B 0,C 180,E1 -20746.341,E2 -20746.341} C_VEL
LIN {X 0,Y 214.004,Z 354.833,A -85,B 0,C 180,E1 -20749.055,E2 -20749.055} C_VEL
LIN {X 0,Y 214.159,Z 356.651,A -85,B 0,C 180,E1 -20751.962,E2 -20751.962} C_VEL
LIN {X 0,Y 214.146,Z 358.607,A -85,B 0,C 180,E1 -20754.748,E2 -20754.748} C_VEL
LIN {X 0,Y 215.269,Z 361.734,A -85,B 0,C 180,E1 -20755.15,E2 -20755.15} C_VEL
LIN {X 0,Y 219.186,Z 371.392,A -85,B 0,C 180,E1 -20756.582,E2 -20756.582} C_VEL
LIN {X 0,Y 222.802,Z 383.112,A -85,B 0,C 180,E1 -20758.395,E2 -20758.395} C_VEL
LIN {X 0,Y 225.313,Z 395.159,A -85,B 0,C 180,E1 -20760.407,E2 -20760.407} C_VEL
LIN {X 0,Y 226.537,Z 405.175,A -85,B 0,C 180,E1 -20762.268,E2 -20762.268} C_VEL
LIN {X 0,Y 226.735,Z 409.048,A -85,B 0,C 180,E1 -20763.044,E2 -20763.044} C_VEL
LIN {X 0,Y 224.262,Z 419.253,A -85,B 0,C 180,E1 -20764.973,E2 -20764.973} C_VEL
LIN {X 0,Y 221.798,Z 428.855,A -85,B 0,C 180,E1 -20767.298,E2 -20767.298} C_VEL
LIN {X 0,Y 219.2,Z 437.308,A -85,B 0,C 180,E1 -20769.84,E2 -20769.84} C_VEL
LIN {X 0,Y 216.894,Z 444.471,A -85,B 0,C 180,E1 -20772.56,E2 -20772.56} C_VEL
LIN {X 0,Y 215.352,Z 449.296,A -85,B 0,C 180,E1 -20774.867,E2 -20774.867} C_VEL
LIN {X 0,Y 213.84,Z 453.985,A -85,B 0,C 180,E1 -20777.666,E2 -20777.666} C_VEL
LIN {X 0,Y 212.767,Z 457.57,A -85,B 0,C 180,E1 -20780.495,E2 -20780.495} C_VEL
LIN {X 0,Y 212.009,Z 460.623,A -85,B 0,C 180,E1 -20783.982,E2 -20783.982} C_VEL
LIN {X 0,Y 211.71,Z 461.796,A -85,B 0,C 180,E1 -20786.194,E2 -20786.194} C_VEL
LIN {X 0,Y 211.618,Z 462.402,A -85,B 0,C 180,E1 -20788.098,E2 -20788.098} C_VEL
LIN {X 0,Y 211.583,Z 462.629,A -85,B 0,C 180,E1 -20790.001,E2 -20790.001} C_VEL
LIN {X 0,Y 211.616,Z 462.434,A -85,B 0,C 180,E1 -20791.904,E2 -20791.904} C_VEL
LIN {X 0,Y 211.933,Z 460.883,A -85,B 0,C 180,E1 -20795.71,E2 -20795.71} C_VEL
LIN {X 0,Y 212.307,Z 459.525,A -85,B 0,C 180,E1 -20797.61,E2 -20797.61} C_VEL
LIN {X 0,Y 213.065,Z 456.66,A -85,B 0,C 180,E1 -20800.453,E2 -20800.453} C_VEL
LIN {X 0,Y 214.254,Z 452.77,A -85,B 0,C 180,E1 -20803.275,E2 -20803.275} C_VEL
LIN {X 0,Y 215.904,Z 447.748,A -85,B 0,C 180,E1 -20806.063,E2 -20806.063} C_VEL
LIN {X 0,Y 217.91,Z 441.424,A -85,B 0,C 180,E1 -20808.816,E2 -20808.816} C_VEL
LIN {X 0,Y 220.456,Z 433.505,A -85,B 0,C 180,E1 -20811.507,E2 -20811.507} C_VEL
LIN {X 0,Y 222.372,Z 426.902,A -85,B 0,C 180,E1 -20813.355,E2 -20813.355} C_VEL
LIN {X 0,Y 224.708,Z 417.719,A -85,B 0,C 180,E1 -20815.471,E2 -20815.471} C_VEL
LIN {X 0,Y 226.69,Z 409.752,A -85,B 0,C 180,E1 -20816.963,E2 -20816.963} C_VEL
LIN {X 0,Y 226.279,Z 401.861,A -85,B 0,C 180,E1 -20818.499,E2 -20818.499} C_VEL
LIN {X 0,Y 224.715,Z 391.634,A -85,B 0,C 180,E1 -20820.346,E2 -20820.346} C_VEL
LIN {X 0,Y 222.04,Z 380.227,A -85,B 0,C 180,E1 -20822.211,E2 -20822.211} C_VEL
LIN {X 0,Y 218.196,Z 368.66,A -85,B 0,C 180,E1 -20823.971,E2 -20823.971} C_VEL
LIN {X 0,Y 215.238,Z 361.681,A -85,B 0,C 180,E1 -20825.01,E2 -20825.01} C_VEL
LIN {X 0,Y 214.106,Z 358.504,A -85,B 0,C 180,E1 -20825.432,E2 -20825.432} C_VEL
LIN {X 0,Y 214.137,Z 356.411,A -85,B 0,C 180,E1 -20828.578,E2 -20828.578} C_VEL
LIN {X 0,Y 213.993,Z 354.869,A -85,B 0,C 180,E1 -20831.06,E2 -20831.06} C_VEL
LIN {X 0,Y 213.777,Z 353.337,A -85,B 0,C 180,E1 -20833.675,E2 -20833.675} C_VEL
LIN {X 0,Y 213.702,Z 352.868,A -85,B 0,C 180,E1 -20836.345,E2 -20836.345} C_VEL
LIN {X 0,Y 213.703,Z 352.866,A -85,B 0,C 180,E1 -20841.329,E2 -20841.329} C_VEL
LIN {X 0,Y 213.754,Z 352.859,A -85,B 0,C 180,E1 -20846.017,E2 -20846.017} C_VEL
LIN {X 0,Y 213.75,Z 352.859,A -85,B 0,C 180,E1 -20850.449,E2 -20850.449} C_VEL
LIN {X 0,Y 213.781,Z 352.852,A -85,B 0,C 180,E1 -20854.699,E2 -20854.699} C_VEL
LIN {X 0,Y 213.806,Z 352.853,A -85,B 0,C 180,E1 -20858.802,E2 -20858.802} C_VEL
LIN {X 0,Y 213.944,Z 352.835,A -85,B 0,C 180,E1 -20862.803,E2 -20862.803} C_VEL
LIN {X 0,Y 213.954,Z 352.836,A -85,B 0,C 180,E1 -20866.706,E2 -20866.706} C_VEL
LIN {X 0,Y 214.168,Z 352.807,A -85,B 0,C 180,E1 -20870.556,E2 -20870.556} C_VEL
LIN {X 0,Y 214.227,Z 352.801,A -85,B 0,C 180,E1 -20872.459,E2 -20872.459} C_VEL
LIN {X 0,Y 214.443,Z 352.773,A -85,B 0,C 180,E1 -20878.122,E2 -20878.122} C_VEL
LIN {X 0,Y 214.534,Z 352.762,A -85,B 0,C 180,E1 -20880,E2 -20880} C_VEL
LIN {X 0,Y 214.443,Z 352.772,A -85,B 0,C 180,E1 -20881.878,E2 -20881.878} C_VEL
LIN {X 0,Y 214.198,Z 352.805,A -85,B 0,C 180,E1 -20887.541,E2 -20887.541} C_VEL
LIN {X 0,Y 213.999,Z 352.829,A -85,B 0,C 180,E1 -20891.364,E2 -20891.364} C_VEL
LIN {X 0,Y 213.932,Z 352.839,A -85,B 0,C 180,E1 -20895.237,E2 -20895.237} C_VEL
LIN {X 0,Y 213.837,Z 352.85,A -85,B 0,C 180,E1 -20899.188,E2 -20899.188} C_VEL
LIN {X 0,Y 213.802,Z 352.854,A -85,B 0,C 180,E1 -20903.232,E2 -20903.232} C_VEL
LIN {X 0,Y 213.786,Z 352.856,A -85,B 0,C 180,E1 -20907.428,E2 -20907.428} C_VEL
LIN {X 0,Y 213.758,Z 352.862,A -85,B 0,C 180,E1 -20911.739,E2 -20911.739} C_VEL
LIN {X 0,Y 213.766,Z 352.889,A -85,B 0,C 180,E1 -20914.722,E2 -20914.722} C_VEL
LIN {X 0,Y 214.18,Z 355.437,A -85,B 0,C 180,E1 -20918.569,E2 -20918.569} C_VEL
LIN {X 0,Y 214.469,Z 357.216,A -85,B 0,C 180,E1 -20921.089,E2 -20921.089} C_VEL
LIN {X 0,Y 215.141,Z 360.911,A -85,B 0,C 180,E1 -20925.945,E2 -20925.945} C_VEL
LIN {X 0,Y 215.629,Z 363.648,A -85,B 0,C 180,E1 -20929.318,E2 -20929.318} C_VEL
LIN {X 0,Y 215.694,Z 366.805,A -85,B 0,C 180,E1 -20932.93,E2 -20932.93} C_VEL
LIN {X 0,Y 215.523,Z 368.613,A -85,B 0,C 180,E1 -20934.874,E2 -20934.874} C_VEL
LIN {X 0,Y 216.627,Z 372.12,A -85,B 0,C 180,E1 -20935.275,E2 -20935.275} C_VEL
LIN {X 0,Y 220.3,Z 384.722,A -85,B 0,C 180,E1 -20936.869,E2 -20936.869} C_VEL
LIN {X 0,Y 222.645,Z 396.215,A -85,B 0,C 180,E1 -20938.461,E2 -20938.461} C_VEL
LIN {X 0,Y 224.031,Z 406.859,A -85,B 0,C 180,E1 -20940.107,E2 -20940.107} C_VEL
LIN {X 0,Y 224.621,Z 417.769,A -85,B 0,C 180,E1 -20942.009,E2 -20942.009} C_VEL
LIN {X 0,Y 224.603,Z 422.96,A -85,B 0,C 180,E1 -20943.017,E2 -20943.017} C_VEL
LIN {X 0,Y 223.97,Z 425.626,A -85,B 0,C 180,E1 -20943.502,E2 -20943.502} C_VEL
LIN {X 0,Y 221.747,Z 429.226,A -85,B 0,C 180,E1 -20944.038,E2 -20944.038} C_VEL
LIN {X 0,Y 216.139,Z 435.873,A -85,B 0,C 180,E1 -20945.067,E2 -20945.067} C_VEL
LIN {X 0,Y 214.66,Z 438.716,A -85,B 0,C 180,E1 -20945.71,E2 -20945.71} C_VEL
LIN {X 0,Y 212.214,Z 447.276,A -85,B 0,C 180,E1 -20948.207,E2 -20948.207} C_VEL
LIN {X 0,Y 209.721,Z 454.731,A -85,B 0,C 180,E1 -20950.929,E2 -20950.929} C_VEL
LIN {X 0,Y 208.071,Z 460.004,A -85,B 0,C 180,E1 -20953.315,E2 -20953.315} C_VEL
LIN {X 0,Y 206.429,Z 465.113,A -85,B 0,C 180,E1 -20956.212,E2 -20956.212} C_VEL
LIN {X 0,Y 205.394,Z 469.088,A -85,B 0,C 180,E1 -20959.152,E2 -20959.152} C_VEL
LIN {X 0,Y 204.68,Z 472.026,A -85,B 0,C 180,E1 -20962.105,E2 -20962.105} C_VEL
LIN {X 0,Y 204.358,Z 474.327,A -85,B 0,C 180,E1 -20965.813,E2 -20965.813} C_VEL
LIN {X 0,Y 204.364,Z 475.039,A -85,B 0,C 180,E1 -20968.028,E2 -20968.028} C_VEL
LIN {X 0,Y 204.451,Z 475.256,A -85,B 0,C 180,E1 -20969.999,E2 -20969.999} C_VEL
LIN {X 0,Y 204.364,Z 475.031,A -85,B 0,C 180,E1 -20971.97,E2 -20971.97} C_VEL
LIN {X 0,Y 204.358,Z 474.314,A -85,B 0,C 180,E1 -20974.186,E2 -20974.186} C_VEL
LIN {X 0,Y 204.679,Z 471.998,A -85,B 0,C 180,E1 -20977.893,E2 -20977.893} C_VEL
LIN {X 0,Y 205.393,Z 469.047,A -85,B 0,C 180,E1 -20980.846,E2 -20980.846} C_VEL
LIN {X 0,Y 206.428,Z 465.055,A -85,B 0,C 180,E1 -20983.786,E2 -20983.786} C_VEL
LIN {X 0,Y 208.366,Z 458.927,A -85,B 0,C 180,E1 -20987.164,E2 -20987.164} C_VEL
LIN {X 0,Y 210.548,Z 452.24,A -85,B 0,C 180,E1 -20990.006,E2 -20990.006} C_VEL
LIN {X 0,Y 212.672,Z 445.235,A -85,B 0,C 180,E1 -20992.403,E2 -20992.403} C_VEL
LIN {X 0,Y 215.002,Z 437.241,A -85,B 0,C 180,E1 -20994.63,E2 -20994.63} C_VEL
LIN {X 0,Y 217.787,Z 427.254,A -85,B 0,C 180,E1 -20996.856,E2 -20996.856} C_VEL
LIN {X 0,Y 217.992,Z 417.316,A -85,B 0,C 180,E1 -20998.919,E2 -20998.919} C_VEL
LIN {X 0,Y 217.456,Z 406.501,A -85,B 0,C 180,E1 -21000.866,E2 -21000.866} C_VEL
LIN {X 0,Y 215.966,Z 395.461,A -85,B 0,C 180,E1 -21002.645,E2 -21002.645} C_VEL
LIN {X 0,Y 213.386,Z 383.588,A -85,B 0,C 180,E1 -21004.379,E2 -21004.379} C_VEL
LIN {X 0,Y 210.118,Z 372.596,A -85,B 0,C 180,E1 -21005.861,E2 -21005.861} C_VEL
LIN {X 0,Y 208.729,Z 369.107,A -85,B 0,C 180,E1 -21006.354,E2 -21006.354} C_VEL
LIN {X 0,Y 208.603,Z 368.266,A -85,B 0,C 180,E1 -21006.493,E2 -21006.493} C_VEL
LIN {X 0,Y 208.676,Z 365.445,A -85,B 0,C 180,E1 -21009.782,E2 -21009.782} C_VEL
LIN {X 0,Y 208.392,Z 363.341,A -85,B 0,C 180,E1 -21012.413,E2 -21012.413} C_VEL
LIN {X 0,Y 207.67,Z 359.584,A -85,B 0,C 180,E1 -21017.402,E2 -21017.402} C_VEL
LIN {X 0,Y 207.109,Z 356.159,A -85,B 0,C 180,E1 -21022.352,E2 -21022.352} C_VEL
LIN {X 0,Y 206.684,Z 353.741,A -85,B 0,C 180,E1 -21026.457,E2 -21026.457} C_VEL
LIN {X 0,Y 206.69,Z 353.74,A -85,B 0,C 180,E1 -21029.333,E2 -21029.333} C_VEL
LIN {X 0,Y 206.699,Z 353.74,A -85,B 0,C 180,E1 -21033.768,E2 -21033.768} C_VEL
LIN {X 0,Y 206.731,Z 353.734,A -85,B 0,C 180,E1 -21038.04,E2 -21038.04} C_VEL
LIN {X 0,Y 206.867,Z 353.717,A -85,B 0,C 180,E1 -21042.196,E2 -21042.196} C_VEL
LIN {X 0,Y 206.906,Z 353.712,A -85,B 0,C 180,E1 -21046.245,E2 -21046.245} C_VEL
LIN {X 0,Y 207.1,Z 353.689,A -85,B 0,C 180,E1 -21050.231,E2 -21050.231} C_VEL
LIN {X 0,Y 207.162,Z 353.681,A -85,B 0,C 180,E1 -21052.201,E2 -21052.201} C_VEL
LIN {X 0,Y 207.376,Z 353.654,A -85,B 0,C 180,E1 -21058.058,E2 -21058.058} C_VEL
LIN {X 0,Y 207.495,Z 353.638,A -85,B 0,C 180,E1 -21060,E2 -21060} C_VEL
LIN {X 0,Y 207.375,Z 353.652,A -85,B 0,C 180,E1 -21061.942,E2 -21061.942} C_VEL
LIN {X 0,Y 207.182,Z 353.676,A -85,B 0,C 180,E1 -21067.798,E2 -21067.798} C_VEL
LIN {X 0,Y 206.94,Z 353.707,A -85,B 0,C 180,E1 -21071.758,E2 -21071.758} C_VEL
LIN {X 0,Y 206.861,Z 353.717,A -85,B 0,C 180,E1 -21075.771,E2 -21075.771} C_VEL
LIN {X 0,Y 206.774,Z 353.727,A -85,B 0,C 180,E1 -21079.87,E2 -21079.87} C_VEL
LIN {X 0,Y 206.733,Z 353.732,A -85,B 0,C 180,E1 -21084.076,E2 -21084.076} C_VEL
LIN {X 0,Y 206.683,Z 353.74,A -85,B 0,C 180,E1 -21088.428,E2 -21088.428} C_VEL
LIN {X 0,Y 206.69,Z 353.739,A -85,B 0,C 180,E1 -21092.959,E2 -21092.959} C_VEL
LIN {X 0,Y 206.669,Z 353.741,A -85,B 0,C 180,E1 -21097.743,E2 -21097.743} C_VEL
LIN {X 0,Y 206.628,Z 353.745,A -85,B 0,C 180,E1 -21101.561,E2 -21101.561} C_VEL
LIN {X 0,Y 206.617,Z 353.749,A -85,B 0,C 180,E1 -21104.416,E2 -21104.416} C_VEL
LIN {X 0,Y 206.829,Z 355.026,A -85,B 0,C 180,E1 -21107.19,E2 -21107.19} C_VEL
LIN {X 0,Y 207.136,Z 357.445,A -85,B 0,C 180,E1 -21111.295,E2 -21111.295} C_VEL
LIN {X 0,Y 207.129,Z 358.727,A -85,B 0,C 180,E1 -21113.334,E2 -21113.334} C_VEL
LIN {X 0,Y 208.375,Z 362.054,A -85,B 0,C 180,E1 -21113.822,E2 -21113.822} C_VEL
LIN {X 0,Y 212.02,Z 370.512,A -85,B 0,C 180,E1 -21115.185,E2 -21115.185} C_VEL
LIN {X 0,Y 215.709,Z 381.771,A -85,B 0,C 180,E1 -21117.03,E2 -21117.03} C_VEL
LIN {X 0,Y 218.275,Z 393.074,A -85,B 0,C 180,E1 -21118.993,E2 -21118.993} C_VEL
LIN {X 0,Y 219.832,Z 404.047,A -85,B 0,C 180,E1 -21121.093,E2 -21121.093} C_VEL
LIN {X 0,Y 220.154,Z 410.544,A -85,B 0,C 180,E1 -21122.428,E2 -21122.428} C_VEL
LIN {X 0,Y 217.843,Z 419.473,A -85,B 0,C 180,E1 -21124.182,E2 -21124.182} C_VEL
LIN {X 0,Y 215.216,Z 429.209,A -85,B 0,C 180,E1 -21126.605,E2 -21126.605} C_VEL
LIN {X 0,Y 212.549,Z 437.525,A -85,B 0,C 180,E1 -21129.18,E2 -21129.18} C_VEL
LIN {X 0,Y 210.125,Z 444.688,A -85,B 0,C 180,E1 -21131.979,E2 -21131.979} C_VEL
LIN {X 0,Y 208.514,Z 449.513,A -85,B 0,C 180,E1 -21134.358,E2 -21134.358} C_VEL
LIN {X 0,Y 206.904,Z 454.202,A -85,B 0,C 180,E1 -21137.246,E2 -21137.246} C_VEL
LIN {X 0,Y 205.753,Z 457.787,A -85,B 0,C 180,E1 -21140.167,E2 -21140.167} C_VEL
LIN {X 0,Y 205.27,Z 459.635,A -85,B 0,C 180,E1 -21142.13,E2 -21142.13} C_VEL
LIN {X 0,Y 204.9,Z 461.023,A -85,B 0,C 180,E1 -21144.095,E2 -21144.095} C_VEL
LIN {X 0,Y 204.521,Z 462.618,A -85,B 0,C 180,E1 -21148.032,E2 -21148.032} C_VEL
LIN {X 0,Y 204.502,Z 462.844,A -85,B 0,C 180,E1 -21150.001,E2 -21150.001} C_VEL
LIN {X 0,Y 204.519,Z 462.65,A -85,B 0,C 180,E1 -21151.97,E2 -21151.97} C_VEL
LIN {X 0,Y 204.864,Z 461.098,A -85,B 0,C 180,E1 -21155.908,E2 -21155.908} C_VEL
LIN {X 0,Y 205.274,Z 459.74,A -85,B 0,C 180,E1 -21157.872,E2 -21157.872} C_VEL
LIN {X 0,Y 206.081,Z 456.874,A -85,B 0,C 180,E1 -21160.812,E2 -21160.812} C_VEL
LIN {X 0,Y 207.344,Z 452.984,A -85,B 0,C 180,E1 -21163.726,E2 -21163.726} C_VEL
LIN {X 0,Y 209.064,Z 447.963,A -85,B 0,C 180,E1 -21166.604,E2 -21166.604} C_VEL
LIN {X 0,Y 211.218,Z 441.637,A -85,B 0,C 180,E1 -21169.435,E2 -21169.435} C_VEL
LIN {X 0,Y 213.86,Z 433.718,A -85,B 0,C 180,E1 -21172.205,E2 -21172.205} C_VEL
LIN {X 0,Y 216.083,Z 426.003,A -85,B 0,C 180,E1 -21174.399,E2 -21174.399} C_VEL
LIN {X 0,Y 218.61,Z 416.865,A -85,B 0,C 180,E1 -21176.492,E2 -21176.492} C_VEL
LIN {X 0,Y 220.259,Z 409.967,A -85,B 0,C 180,E1 -21177.818,E2 -21177.818} C_VEL
LIN {X 0,Y 219.411,Z 399.963,A -85,B 0,C 180,E1 -21179.854,E2 -21179.854} C_VEL
LIN {X 0,Y 217.357,Z 388.34,A -85,B 0,C 180,E1 -21181.989,E2 -21181.989} C_VEL
LIN {X 0,Y 214.348,Z 377.2,A -85,B 0,C 180,E1 -21183.876,E2 -21183.876} C_VEL
LIN {X 0,Y 210.296,Z 366.131,A -85,B 0,C 180,E1 -21185.661,E2 -21185.661} C_VEL
LIN {X 0,Y 208.072,Z 361.526,A -85,B 0,C 180,E1 -21186.431,E2 -21186.431} C_VEL
LIN {X 0,Y 207.139,Z 358.723,A -85,B 0,C 180,E1 -21186.837,E2 -21186.837} C_VEL
LIN {X 0,Y 207.032,Z 356.673,A -85,B 0,C 180,E1 -21190.164,E2 -21190.164} C_VEL
LIN {X 0,Y 206.707,Z 354.228,A -85,B 0,C 180,E1 -21194.439,E2 -21194.439} C_VEL
LIN {X 0,Y 206.618,Z 353.751,A -85,B 0,C 180,E1 -21195.586,E2 -21195.586} C_VEL
LIN {X 0,Y 206.647,Z 353.745,A -85,B 0,C 180,E1 -21199.745,E2 -21199.745} C_VEL
LIN {X 0,Y 206.7,Z 353.737,A -85,B 0,C 180,E1 -21204.689,E2 -21204.689} C_VEL
LIN {X 0,Y 206.696,Z 353.74,A -85,B 0,C 180,E1 -21209.334,E2 -21209.334} C_VEL
LIN {X 0,Y 206.705,Z 353.735,A -85,B 0,C 180,E1 -21213.768,E2 -21213.768} C_VEL
LIN {X 0,Y 206.737,Z 353.731,A -85,B 0,C 180,E1 -21218.041,E2 -21218.041} C_VEL
LIN {X 0,Y 206.873,Z 353.716,A -85,B 0,C 180,E1 -21222.196,E2 -21222.196} C_VEL
LIN {X 0,Y 206.896,Z 353.713,A -85,B 0,C 180,E1 -21226.244,E2 -21226.244} C_VEL
LIN {X 0,Y 207.106,Z 353.687,A -85,B 0,C 180,E1 -21230.231,E2 -21230.231} C_VEL
LIN {X 0,Y 207.168,Z 353.68,A -85,B 0,C 180,E1 -21232.201,E2 -21232.201} C_VEL
LIN {X 0,Y 207.38,Z 353.653,A -85,B 0,C 180,E1 -21238.058,E2 -21238.058} C_VEL
LIN {X 0,Y 207.5,Z 353.639,A -85,B 0,C 180,E1 -21240,E2 -21240} C_VEL
LIN {X 0,Y 207.379,Z 353.652,A -85,B 0,C 180,E1 -21241.942,E2 -21241.942} C_VEL
LIN {X 0,Y 207.14,Z 353.685,A -85,B 0,C 180,E1 -21247.8,E2 -21247.8} C_VEL
LIN {X 0,Y 206.924,Z 353.711,A -85,B 0,C 180,E1 -21251.758,E2 -21251.758} C_VEL
LIN {X 0,Y 206.866,Z 353.719,A -85,B 0,C 180,E1 -21255.771,E2 -21255.771} C_VEL
LIN {X 0,Y 206.78,Z 353.729,A -85,B 0,C 180,E1 -21259.869,E2 -21259.869} C_VEL
LIN {X 0,Y 206.738,Z 353.733,A -85,B 0,C 180,E1 -21264.075,E2 -21264.075} C_VEL
LIN {X 0,Y 206.688,Z 353.741,A -85,B 0,C 180,E1 -21268.427,E2 -21268.427} C_VEL
LIN {X 0,Y 206.694,Z 353.742,A -85,B 0,C 180,E1 -21272.959,E2 -21272.959} C_VEL
LIN {X 0,Y 206.765,Z 353.995,A -85,B 0,C 180,E1 -21274.114,E2 -21274.114} C_VEL
LIN {X 0,Y 207.227,Z 356.958,A -85,B 0,C 180,E1 -21278.736,E2 -21278.736} C_VEL
LIN {X 0,Y 207.66,Z 359.638,A -85,B 0,C 180,E1 -21282.6,E2 -21282.6} C_VEL
LIN {X 0,Y 208.352,Z 363.387,A -85,B 0,C 180,E1 -21287.575,E2 -21287.575} C_VEL
LIN {X 0,Y 208.661,Z 365.96,A -85,B 0,C 180,E1 -21290.776,E2 -21290.776} C_VEL
LIN {X 0,Y 208.623,Z 368.454,A -85,B 0,C 180,E1 -21293.533,E2 -21293.533} C_VEL
LIN {X 0,Y 209.58,Z 371.611,A -85,B 0,C 180,E1 -21293.912,E2 -21293.912} C_VEL
LIN {X 0,Y 211.758,Z 377.658,A -85,B 0,C 180,E1 -21294.758,E2 -21294.758} C_VEL
LIN {X 0,Y 214.684,Z 388.719,A -85,B 0,C 180,E1 -21296.308,E2 -21296.308} C_VEL
LIN {X 0,Y 216.831,Z 400.854,A -85,B 0,C 180,E1 -21298.155,E2 -21298.155} C_VEL
LIN {X 0,Y 217.914,Z 412.332,A -85,B 0,C 180,E1 -21300.113,E2 -21300.113} C_VEL
LIN {X 0,Y 218.038,Z 422.74,A -85,B 0,C 180,E1 -21302.136,E2 -21302.136} C_VEL
LIN {X 0,Y 217.609,Z 428.507,A -85,B 0,C 180,E1 -21303.377,E2 -21303.377} C_VEL
LIN {X 0,Y 214.66,Z 438.716,A -85,B 0,C 180,E1 -21305.71,E2 -21305.71} C_VEL
LIN {X 0,Y 212.89,Z 442.806,A -85,B 0,C 180,E1 -21306.751,E2 -21306.751} C_VEL
LIN {X 0,Y 208.306,Z 449.014,A -85,B 0,C 180,E1 -21308.449,E2 -21308.449} C_VEL
LIN {X 0,Y 203.722,Z 454.581,A -85,B 0,C 180,E1 -21310.351,E2 -21310.351} C_VEL
LIN {X 0,Y 201.993,Z 457.668,A -85,B 0,C 180,E1 -21311.693,E2 -21311.693} C_VEL
LIN {X 0,Y 200.021,Z 463.306,A -85,B 0,C 180,E1 -21314.72,E2 -21314.72} C_VEL
LIN {X 0,Y 198.705,Z 467.646,A -85,B 0,C 180,E1 -21317.747,E2 -21317.747} C_VEL
LIN {X 0,Y 198.092,Z 469.947,A -85,B 0,C 180,E1 -21319.781,E2 -21319.781} C_VEL
LIN {X 0,Y 197.646,Z 471.811,A -85,B 0,C 180,E1 -21321.822,E2 -21321.822} C_VEL
LIN {X 0,Y 197.368,Z 473.21,A -85,B 0,C 180,E1 -21323.867,E2 -21323.867} C_VEL
LIN {X 0,Y 197.246,Z 474.278,A -85,B 0,C 180,E1 -21326.08,E2 -21326.08} C_VEL
LIN {X 0,Y 197.27,Z 474.824,A -85,B 0,C 180,E1 -21327.957,E2 -21327.957} C_VEL
LIN {X 0,Y 197.352,Z 475.041,A -85,B 0,C 180,E1 -21329.999,E2 -21329.999} C_VEL
LIN {X 0,Y 197.245,Z 474.264,A -85,B 0,C 180,E1 -21333.918,E2 -21333.918} C_VEL
LIN {X 0,Y 197.368,Z 473.191,A -85,B 0,C 180,E1 -21336.131,E2 -21336.131} C_VEL
LIN {X 0,Y 197.645,Z 471.782,A -85,B 0,C 180,E1 -21338.176,E2 -21338.176} C_VEL
LIN {X 0,Y 198.38,Z 468.829,A -85,B 0,C 180,E1 -21341.235,E2 -21341.235} C_VEL
LIN {X 0,Y 199.495,Z 464.837,A -85,B 0,C 180,E1 -21344.275,E2 -21344.275} C_VEL
LIN {X 0,Y 201.58,Z 458.71,A -85,B 0,C 180,E1 -21347.761,E2 -21347.761} C_VEL
LIN {X 0,Y 203.886,Z 452.022,A -85,B 0,C 180,E1 -21350.689,E2 -21350.689} C_VEL
LIN {X 0,Y 206.447,Z 443.801,A -85,B 0,C 180,E1 -21353.549,E2 -21353.549} C_VEL
LIN {X 0,Y 209.113,Z 435.218,A -85,B 0,C 180,E1 -21355.906,E2 -21355.906} C_VEL
LIN {X 0,Y 211.146,Z 428.107,A -85,B 0,C 180,E1 -21357.504,E2 -21357.504} C_VEL
LIN {X 0,Y 211.468,Z 418.439,A -85,B 0,C 180,E1 -21359.621,E2 -21359.621} C_VEL
LIN {X 0,Y 211.065,Z 407.989,A -85,B 0,C 180,E1 -21361.628,E2 -21361.628} C_VEL
LIN {X 0,Y 209.634,Z 396.322,A -85,B 0,C 180,E1 -21363.622,E2 -21363.622} C_VEL
LIN {X 0,Y 207.093,Z 384.522,A -85,B 0,C 180,E1 -21365.465,E2 -21365.465} C_VEL
LIN {X 0,Y 204.504,Z 375.71,A -85,B 0,C 180,E1 -21366.771,E2 -21366.771} C_VEL
LIN {X 0,Y 201.736,Z 368.615,A -85,B 0,C 180,E1 -21367.841,E2 -21367.841} C_VEL
LIN {X 0,Y 201.671,Z 368.043,A -85,B 0,C 180,E1 -21367.916,E2 -21367.916} C_VEL
LIN {X 0,Y 201.475,Z 365.188,A -85,B 0,C 180,E1 -21371.509,E2 -21371.509} C_VEL
LIN {X 0,Y 200.93,Z 362.148,A -85,B 0,C 180,E1 -21375.609,E2 -21375.609} C_VEL
LIN {X 0,Y 200.327,Z 358.766,A -85,B 0,C 180,E1 -21380.515,E2 -21380.515} C_VEL
LIN {X 0,Y 199.812,Z 355.507,A -85,B 0,C 180,E1 -21385.752,E2 -21385.752} C_VEL
LIN {X 0,Y 199.641,Z 354.619,A -85,B 0,C 180,E1 -21387.655,E2 -21387.655} C_VEL
LIN {X 0,Y 199.637,Z 354.619,A -85,B 0,C 180,E1 -21392.764,E2 -21392.764} C_VEL
LIN {X 0,Y 199.703,Z 354.61,A -85,B 0,C 180,E1 -21397.225,E2 -21397.225} C_VEL
LIN {X 0,Y 199.791,Z 354.599,A -85,B 0,C 180,E1 -21401.758,E2 -21401.758} C_VEL
LIN {X 0,Y 199.841,Z 354.594,A -85,B 0,C 180,E1 -21405.749,E2 -21405.749} C_VEL
LIN {X 0,Y 200.065,Z 354.564,A -85,B 0,C 180,E1 -21409.884,E2 -21409.884} C_VEL
LIN {X 0,Y 200.03,Z 354.568,A -85,B 0,C 180,E1 -21413.95,E2 -21413.95} C_VEL
LIN {X 0,Y 200.315,Z 354.534,A -85,B 0,C 180,E1 -21417.989,E2 -21417.989} C_VEL
LIN {X 0,Y 200.461,Z 354.514,A -85,B 0,C 180,E1 -21420,E2 -21420} C_VEL
LIN {X 0,Y 200.025,Z 354.569,A -85,B 0,C 180,E1 -21424.03,E2 -21424.03} C_VEL
LIN {X 0,Y 200.126,Z 354.554,A -85,B 0,C 180,E1 -21428.075,E2 -21428.075} C_VEL
LIN {X 0,Y 200.063,Z 354.564,A -85,B 0,C 180,E1 -21430.398,E2 -21430.398} C_VEL
LIN {X 0,Y 199.799,Z 354.596,A -85,B 0,C 180,E1 -21436.344,E2 -21436.344} C_VEL
LIN {X 0,Y 199.685,Z 354.611,A -85,B 0,C 180,E1 -21440.607,E2 -21440.607} C_VEL
LIN {X 0,Y 199.645,Z 354.616,A -85,B 0,C 180,E1 -21444.988,E2 -21444.988} C_VEL
LIN {X 0,Y 199.603,Z 354.622,A -85,B 0,C 180,E1 -21449.534,E2 -21449.534} C_VEL
LIN {X 0,Y 199.661,Z 354.615,A -85,B 0,C 180,E1 -21452.354,E2 -21452.354} C_VEL
LIN {X 0,Y 199.615,Z 354.621,A -85,B 0,C 180,E1 -21456.765,E2 -21456.765} C_VEL
LIN {X 0,Y 199.591,Z 354.623,A -85,B 0,C 180,E1 -21459.332,E2 -21459.332} C_VEL
LIN {X 0,Y 199.563,Z 354.628,A -85,B 0,C 180,E1 -21462.309,E2 -21462.309} C_VEL
LIN {X 0,Y 199.696,Z 355.294,A -85,B 0,C 180,E1 -21465.264,E2 -21465.264} C_VEL
LIN {X 0,Y 199.95,Z 356.823,A -85,B 0,C 180,E1 -21468.103,E2 -21468.103} C_VEL
LIN {X 0,Y 200.136,Z 359.006,A -85,B 0,C 180,E1 -21471.846,E2 -21471.846} C_VEL
LIN {X 0,Y 201.344,Z 362.253,A -85,B 0,C 180,E1 -21472.339,E2 -21472.339} C_VEL
LIN {X 0,Y 202.555,Z 364.593,A -85,B 0,C 180,E1 -21472.767,E2 -21472.767} C_VEL
LIN {X 0,Y 206.479,Z 373.959,A -85,B 0,C 180,E1 -21474.428,E2 -21474.428} C_VEL
LIN {X 0,Y 209.505,Z 383.57,A -85,B 0,C 180,E1 -21476.125,E2 -21476.125} C_VEL
LIN {X 0,Y 211.942,Z 394.609,A -85,B 0,C 180,E1 -21478.167,E2 -21478.167} C_VEL
LIN {X 0,Y 213.173,Z 403.964,A -85,B 0,C 180,E1 -21480.038,E2 -21480.038} C_VEL
LIN {X 0,Y 213.611,Z 411.944,A -85,B 0,C 180,E1 -21481.776,E2 -21481.776} C_VEL
LIN {X 0,Y 210.925,Z 421.644,A -85,B 0,C 180,E1 -21483.803,E2 -21483.803} C_VEL
LIN {X 0,Y 208.369,Z 430.464,A -85,B 0,C 180,E1 -21486.126,E2 -21486.126} C_VEL
LIN {X 0,Y 205.499,Z 439.069,A -85,B 0,C 180,E1 -21488.957,E2 -21488.957} C_VEL
LIN {X 0,Y 202.995,Z 445.931,A -85,B 0,C 180,E1 -21491.846,E2 -21491.846} C_VEL
LIN {X 0,Y 201.051,Z 451.42,A -85,B 0,C 180,E1 -21494.802,E2 -21494.802} C_VEL
LIN {X 0,Y 199.52,Z 455.726,A -85,B 0,C 180,E1 -21497.8,E2 -21497.8} C_VEL
LIN {X 0,Y 198.764,Z 458.003,A -85,B 0,C 180,E1 -21499.818,E2 -21499.818} C_VEL
LIN {X 0,Y 198.232,Z 459.851,A -85,B 0,C 180,E1 -21501.848,E2 -21501.848} C_VEL
LIN {X 0,Y 197.763,Z 461.467,A -85,B 0,C 180,E1 -21504.301,E2 -21504.301} C_VEL
LIN {X 0,Y 197.427,Z 462.833,A -85,B 0,C 180,E1 -21507.961,E2 -21507.961} C_VEL
LIN {X 0,Y 197.424,Z 463.059,A -85,B 0,C 180,E1 -21510.001,E2 -21510.001} C_VEL
LIN {X 0,Y 197.426,Z 462.865,A -85,B 0,C 180,E1 -21512.041,E2 -21512.041} C_VEL
LIN {X 0,Y 197.801,Z 461.313,A -85,B 0,C 180,E1 -21516.12,E2 -21516.12} C_VEL
LIN {X 0,Y 198.237,Z 459.955,A -85,B 0,C 180,E1 -21518.153,E2 -21518.153} C_VEL
LIN {X 0,Y 199.116,Z 457.089,A -85,B 0,C 180,E1 -21521.194,E2 -21521.194} C_VEL
LIN {X 0,Y 200.457,Z 453.198,A -85,B 0,C 180,E1 -21524.207,E2 -21524.207} C_VEL
LIN {X 0,Y 202.254,Z 448.178,A -85,B 0,C 180,E1 -21527.18,E2 -21527.18} C_VEL
LIN {X 0,Y 204.539,Z 441.85,A -85,B 0,C 180,E1 -21530.097,E2 -21530.097} C_VEL
LIN {X 0,Y 207.3,Z 433.931,A -85,B 0,C 180,E1 -21532.947,E2 -21532.947} C_VEL
LIN {X 0,Y 209.502,Z 426.692,A -85,B 0,C 180,E1 -21535.075,E2 -21535.075} C_VEL
LIN {X 0,Y 212.281,Z 417.077,A -85,B 0,C 180,E1 -21537.346,E2 -21537.346} C_VEL
LIN {X 0,Y 213.735,Z 411.402,A -85,B 0,C 180,E1 -21538.476,E2 -21538.476} C_VEL
LIN {X 0,Y 212.971,Z 401.34,A -85,B 0,C 180,E1 -21540.649,E2 -21540.649} C_VEL
LIN {X 0,Y 211.104,Z 390.155,A -85,B 0,C 180,E1 -21542.825,E2 -21542.825} C_VEL
LIN {X 0,Y 208.252,Z 379.251,A -85,B 0,C 180,E1 -21544.8,E2 -21544.8} C_VEL
LIN {X 0,Y 204.607,Z 369.176,A -85,B 0,C 180,E1 -21546.573,E2 -21546.573} C_VEL
LIN {X 0,Y 201.589,Z 362.602,A -85,B 0,C 180,E1 -21547.744,E2 -21547.744} C_VEL
LIN {X 0,Y 200.255,Z 359.521,A -85,B 0,C 180,E1 -21548.257,E2 -21548.257} C_VEL
LIN {X 0,Y 200.165,Z 359.002,A -85,B 0,C 180,E1 -21548.326,E2 -21548.326} C_VEL
LIN {X 0,Y 199.877,Z 356.651,A -85,B 0,C 180,E1 -21552.405,E2 -21552.405} C_VEL
LIN {X 0,Y 199.649,Z 355.132,A -85,B 0,C 180,E1 -21555.248,E2 -21555.248} C_VEL
LIN {X 0,Y 199.571,Z 354.628,A -85,B 0,C 180,E1 -21558.002,E2 -21558.002} C_VEL
LIN {X 0,Y 199.597,Z 354.621,A -85,B 0,C 180,E1 -21560.773,E2 -21560.773} C_VEL
LIN {X 0,Y 199.61,Z 354.62,A -85,B 0,C 180,E1 -21565.713,E2 -21565.713} C_VEL
LIN {X 0,Y 199.686,Z 354.607,A -85,B 0,C 180,E1 -21568.134,E2 -21568.134} C_VEL
LIN {X 0,Y 199.643,Z 354.617,A -85,B 0,C 180,E1 -21572.765,E2 -21572.765} C_VEL
LIN {X 0,Y 199.709,Z 354.609,A -85,B 0,C 180,E1 -21577.225,E2 -21577.225} C_VEL
LIN {X 0,Y 199.797,Z 354.597,A -85,B 0,C 180,E1 -21581.758,E2 -21581.758} C_VEL
LIN {X 0,Y 199.836,Z 354.591,A -85,B 0,C 180,E1 -21585.748,E2 -21585.748} C_VEL
LIN {X 0,Y 200.071,Z 354.563,A -85,B 0,C 180,E1 -21589.884,E2 -21589.884} C_VEL
LIN {X 0,Y 200.034,Z 354.567,A -85,B 0,C 180,E1 -21593.95,E2 -21593.95} C_VEL
LIN {X 0,Y 200.32,Z 354.533,A -85,B 0,C 180,E1 -21597.989,E2 -21597.989} C_VEL
LIN {X 0,Y 200.466,Z 354.515,A -85,B 0,C 180,E1 -21600,E2 -21600} C_VEL
LIN {X 0,Y 200.025,Z 354.569,A -85,B 0,C 180,E1 -21604.029,E2 -21604.029} C_VEL
LIN {X 0,Y 200.089,Z 354.563,A -85,B 0,C 180,E1 -21608.077,E2 -21608.077} C_VEL
LIN {X 0,Y 199.874,Z 354.592,A -85,B 0,C 180,E1 -21612.179,E2 -21612.179} C_VEL
LIN {X 0,Y 199.804,Z 354.599,A -85,B 0,C 180,E1 -21616.344,E2 -21616.344} C_VEL
LIN {X 0,Y 199.691,Z 354.612,A -85,B 0,C 180,E1 -21620.606,E2 -21620.606} C_VEL
LIN {X 0,Y 199.65,Z 354.616,A -85,B 0,C 180,E1 -21624.987,E2 -21624.987} C_VEL
LIN {X 0,Y 199.608,Z 354.623,A -85,B 0,C 180,E1 -21629.533,E2 -21629.533} C_VEL
LIN {X 0,Y 199.683,Z 354.738,A -85,B 0,C 180,E1 -21632.814,E2 -21632.814} C_VEL
LIN {X 0,Y 200.033,Z 357.023,A -85,B 0,C 180,E1 -21636.675,E2 -21636.675} C_VEL
LIN {X 0,Y 200.598,Z 360.341,A -85,B 0,C 180,E1 -21641.734,E2 -21641.734} C_VEL
LIN {X 0,Y 201.059,Z 363.118,A -85,B 0,C 180,E1 -21645.645,E2 -21645.645} C_VEL
LIN {X 0,Y 201.618,Z 366.471,A -85,B 0,C 180,E1 -21650.074,E2 -21650.074} C_VEL
LIN {X 0,Y 201.643,Z 368.139,A -85,B 0,C 180,E1 -21652.049,E2 -21652.049} C_VEL
LIN {X 0,Y 202.658,Z 371.239,A -85,B 0,C 180,E1 -21652.463,E2 -21652.463} C_VEL
LIN {X 0,Y 203.912,Z 374.339,A -85,B 0,C 180,E1 -21652.94,E2 -21652.94} C_VEL
LIN {X 0,Y 206.163,Z 380.787,A -85,B 0,C 180,E1 -21653.929,E2 -21653.929} C_VEL
LIN {X 0,Y 208.786,Z 391.492,A -85,B 0,C 180,E1 -21655.557,E2 -21655.557} C_VEL
LIN {X 0,Y 210.641,Z 403.312,A -85,B 0,C 180,E1 -21657.501,E2 -21657.501} C_VEL
LIN {X 0,Y 211.457,Z 413.877,A -85,B 0,C 180,E1 -21659.435,E2 -21659.435} C_VEL
LIN {X 0,Y 211.4,Z 424.898,A -85,B 0,C 180,E1 -21661.724,E2 -21661.724} C_VEL
LIN {X 0,Y 210.97,Z 429.367,A -85,B 0,C 180,E1 -21662.738,E2 -21662.738} C_VEL
LIN {X 0,Y 208.003,Z 439.104,A -85,B 0,C 180,E1 -21665.062,E2 -21665.062} C_VEL
LIN {X 0,Y 205.839,Z 446.245,A -85,B 0,C 180,E1 -21667.201,E2 -21667.201} C_VEL
LIN {X 0,Y 203.426,Z 453.36,A -85,B 0,C 180,E1 -21669.788,E2 -21669.788} C_VEL
LIN {X 0,Y 201.993,Z 457.668,A -85,B 0,C 180,E1 -21671.693,E2 -21671.693} C_VEL
LIN {X 0,Y 200.347,Z 460.548,A -85,B 0,C 180,E1 -21673.092,E2 -21673.092} C_VEL
LIN {X 0,Y 196.162,Z 464.727,A -85,B 0,C 180,E1 -21675.394,E2 -21675.394} C_VEL
LIN {X 0,Y 192.237,Z 468.169,A -85,B 0,C 180,E1 -21677.883,E2 -21677.883} C_VEL
LIN {X 0,Y 191.041,Z 469.853,A -85,B 0,C 180,E1 -21679.539,E2 -21679.539} C_VEL
LIN {X 0,Y 190.588,Z 471.595,A -85,B 0,C 180,E1 -21681.517,E2 -21681.517} C_VEL
LIN {X 0,Y 190.3,Z 472.995,A -85,B 0,C 180,E1 -21683.638,E2 -21683.638} C_VEL
LIN {X 0,Y 190.138,Z 474.23,A -85,B 0,C 180,E1 -21686.371,E2 -21686.371} C_VEL
LIN {X 0,Y 190.256,Z 474.825,A -85,B 0,C 180,E1 -21689.999,E2 -21689.999} C_VEL
LIN {X 0,Y 190.137,Z 474.215,A -85,B 0,C 180,E1 -21693.628,E2 -21693.628} C_VEL
LIN {X 0,Y 190.3,Z 472.974,A -85,B 0,C 180,E1 -21696.36,E2 -21696.36} C_VEL
LIN {X 0,Y 190.587,Z 471.565,A -85,B 0,C 180,E1 -21698.481,E2 -21698.481} C_VEL
LIN {X 0,Y 191.38,Z 468.612,A -85,B 0,C 180,E1 -21701.651,E2 -21701.651} C_VEL
LIN {X 0,Y 192.583,Z 464.619,A -85,B 0,C 180,E1 -21704.799,E2 -21704.799} C_VEL
LIN {X 0,Y 194.816,Z 458.492,A -85,B 0,C 180,E1 -21708.399,E2 -21708.399} C_VEL
LIN {X 0,Y 197.255,Z 451.805,A -85,B 0,C 180,E1 -21711.418,E2 -21711.418} C_VEL
LIN {X 0,Y 199.937,Z 443.505,A -85,B 0,C 180,E1 -21714.393,E2 -21714.393} C_VEL
LIN {X 0,Y 202.726,Z 434.999,A -85,B 0,C 180,E1 -21716.786,E2 -21716.786} C_VEL
LIN {X 0,Y 204.546,Z 428.96,A -85,B 0,C 180,E1 -21718.191,E2 -21718.191} C_VEL
LIN {X 0,Y 204.969,Z 419.363,A -85,B 0,C 180,E1 -21720.408,E2 -21720.408} C_VEL
LIN {X 0,Y 204.621,Z 408.265,A -85,B 0,C 180,E1 -21722.653,E2 -21722.653} C_VEL
LIN {X 0,Y 203.137,Z 396.132,A -85,B 0,C 180,E1 -21724.842,E2 -21724.842} C_VEL
LIN {X 0,Y 200.594,Z 384.364,A -85,B 0,C 180,E1 -21726.788,E2 -21726.788} C_VEL
LIN {X 0,Y 197.97,Z 376.049,A -85,B 0,C 180,E1 -21728.144,E2 -21728.144} C_VEL
LIN {X 0,Y 195.999,Z 371.578,A -85,B 0,C 180,E1 -21728.937,E2 -21728.937} C_VEL
LIN {X 0,Y 194.783,Z 368.549,A -85,B 0,C 180,E1 -21729.435,E2 -21729.435} C_VEL
LIN {X 0,Y 194.645,Z 367.81,A -85,B 0,C 180,E1 -21729.531,E2 -21729.531} C_VEL
LIN {X 0,Y 194.178,Z 364.774,A -85,B 0,C 180,E1 -21733.625,E2 -21733.625} C_VEL
LIN {X 0,Y 193.814,Z 362.787,A -85,B 0,C 180,E1 -21736.486,E2 -21736.486} C_VEL
LIN {X 0,Y 193.178,Z 359.335,A -85,B 0,C 180,E1 -21741.795,E2 -21741.795} C_VEL
LIN {X 0,Y 192.986,Z 357.777,A -85,B 0,C 180,E1 -21744.361,E2 -21744.361} C_VEL
LIN {X 0,Y 192.596,Z 355.498,A -85,B 0,C 180,E1 -21748.707,E2 -21748.707} C_VEL
LIN {X 0,Y 192.615,Z 355.495,A -85,B 0,C 180,E1 -21751.684,E2 -21751.684} C_VEL
LIN {X 0,Y 192.673,Z 355.485,A -85,B 0,C 180,E1 -21756.344,E2 -21756.344} C_VEL
LIN {X 0,Y 192.726,Z 355.479,A -85,B 0,C 180,E1 -21761.457,E2 -21761.457} C_VEL
LIN {X 0,Y 192.765,Z 355.474,A -85,B 0,C 180,E1 -21765.214,E2 -21765.214} C_VEL
LIN {X 0,Y 192.975,Z 355.446,A -85,B 0,C 180,E1 -21769.508,E2 -21769.508} C_VEL
LIN {X 0,Y 193.056,Z 355.436,A -85,B 0,C 180,E1 -21771.627,E2 -21771.627} C_VEL
LIN {X 0,Y 193.258,Z 355.413,A -85,B 0,C 180,E1 -21777.916,E2 -21777.916} C_VEL
LIN {X 0,Y 193.426,Z 355.39,A -85,B 0,C 180,E1 -21780,E2 -21780} C_VEL
LIN {X 0,Y 192.972,Z 355.447,A -85,B 0,C 180,E1 -21784.177,E2 -21784.177} C_VEL
LIN {X 0,Y 193.073,Z 355.432,A -85,B 0,C 180,E1 -21788.372,E2 -21788.372} C_VEL
LIN {X 0,Y 193.005,Z 355.443,A -85,B 0,C 180,E1 -21790.539,E2 -21790.539} C_VEL
LIN {X 0,Y 192.752,Z 355.474,A -85,B 0,C 180,E1 -21796.959,E2 -21796.959} C_VEL
LIN {X 0,Y 192.615,Z 355.492,A -85,B 0,C 180,E1 -21801.4,E2 -21801.4} C_VEL
LIN {X 0,Y 192.634,Z 355.489,A -85,B 0,C 180,E1 -21804.209,E2 -21804.209} C_VEL
LIN {X 0,Y 192.596,Z 355.494,A -85,B 0,C 180,E1 -21808.867,E2 -21808.867} C_VEL
LIN {X 0,Y 192.59,Z 355.496,A -85,B 0,C 180,E1 -21813.188,E2 -21813.188} C_VEL
LIN {X 0,Y 192.539,Z 355.502,A -85,B 0,C 180,E1 -21818.355,E2 -21818.355} C_VEL
LIN {X 0,Y 192.499,Z 355.576,A -85,B 0,C 180,E1 -21823.1,E2 -21823.1} C_VEL
LIN {X 0,Y 192.816,Z 357.426,A -85,B 0,C 180,E1 -21826.802,E2 -21826.802} C_VEL
LIN {X 0,Y 193.067,Z 359.288,A -85,B 0,C 180,E1 -21830.183,E2 -21830.183} C_VEL
LIN {X 0,Y 194.314,Z 362.487,A -85,B 0,C 180,E1 -21830.717,E2 -21830.717} C_VEL
LIN {X 0,Y 195.567,Z 364.653,A -85,B 0,C 180,E1 -21831.178,E2 -21831.178} C_VEL
LIN {X 0,Y 200.024,Z 374.768,A -85,B 0,C 180,E1 -21833.152,E2 -21833.152} C_VEL
LIN {X 0,Y 203.365,Z 385.399,A -85,B 0,C 180,E1 -21835.17,E2 -21835.17} C_VEL
LIN {X 0,Y 205.61,Z 395.983,A -85,B 0,C 180,E1 -21837.255,E2 -21837.255} C_VEL
LIN {X 0,Y 206.801,Z 405.877,A -85,B 0,C 180,E1 -21839.353,E2 -21839.353} C_VEL
LIN {X 0,Y 207.072,Z 413.332,A -85,B 0,C 180,E1 -21841.078,E2 -21841.078} C_VEL
LIN {X 0,Y 204.57,Z 421.863,A -85,B 0,C 180,E1 -21842.923,E2 -21842.923} C_VEL
LIN {X 0,Y 201.883,Z 430.682,A -85,B 0,C 180,E1 -21845.309,E2 -21845.309} C_VEL
LIN {X 0,Y 199.357,Z 437.961,A -85,B 0,C 180,E1 -21847.731,E2 -21847.731} C_VEL
LIN {X 0,Y 196.681,Z 445.123,A -85,B 0,C 180,E1 -21850.7,E2 -21850.7} C_VEL
LIN {X 0,Y 194.877,Z 449.947,A -85,B 0,C 180,E1 -21853.232,E2 -21853.232} C_VEL
LIN {X 0,Y 193.09,Z 454.635,A -85,B 0,C 180,E1 -21856.316,E2 -21856.316} C_VEL
LIN {X 0,Y 191.773,Z 458.22,A -85,B 0,C 180,E1 -21859.443,E2 -21859.443} C_VEL
LIN {X 0,Y 191.2,Z 460.068,A -85,B 0,C 180,E1 -21861.546,E2 -21861.546} C_VEL
LIN {X 0,Y 190.643,Z 461.885,A -85,B 0,C 180,E1 -21864.474,E2 -21864.474} C_VEL
LIN {X 0,Y 190.336,Z 463.049,A -85,B 0,C 180,E1 -21867.885,E2 -21867.885} C_VEL
LIN {X 0,Y 190.327,Z 463.274,A -85,B 0,C 180,E1 -21870.001,E2 -21870.001} C_VEL
LIN {X 0,Y 190.334,Z 463.08,A -85,B 0,C 180,E1 -21872.117,E2 -21872.117} C_VEL
LIN {X 0,Y 190.739,Z 461.528,A -85,B 0,C 180,E1 -21876.347,E2 -21876.347} C_VEL
LIN {X 0,Y 191.204,Z 460.17,A -85,B 0,C 180,E1 -21878.455,E2 -21878.455} C_VEL
LIN {X 0,Y 192.145,Z 457.304,A -85,B 0,C 180,E1 -21881.606,E2 -21881.606} C_VEL
LIN {X 0,Y 193.59,Z 453.412,A -85,B 0,C 180,E1 -21884.722,E2 -21884.722} C_VEL
LIN {X 0,Y 195.472,Z 448.392,A -85,B 0,C 180,E1 -21887.795,E2 -21887.795} C_VEL
LIN {X 0,Y 197.883,Z 442.063,A -85,B 0,C 180,E1 -21890.804,E2 -21890.804} C_VEL
LIN {X 0,Y 200.775,Z 434.145,A -85,B 0,C 180,E1 -21893.738,E2 -21893.738} C_VEL
LIN {X 0,Y 203.391,Z 425.902,A -85,B 0,C 180,E1 -21896.194,E2 -21896.194} C_VEL
LIN {X 0,Y 206.334,Z 416.222,A -85,B 0,C 180,E1 -21898.481,E2 -21898.481} C_VEL
LIN {X 0,Y 207.238,Z 412.782,A -85,B 0,C 180,E1 -21899.176,E2 -21899.176} C_VEL
LIN {X 0,Y 206.637,Z 403.157,A -85,B 0,C 180,E1 -21901.374,E2 -21901.374} C_VEL
LIN {X 0,Y 204.881,Z 391.964,A -85,B 0,C 180,E1 -21903.711,E2 -21903.711} C_VEL
LIN {X 0,Y 202.269,Z 381.557,A -85,B 0,C 180,E1 -21905.734,E2 -21905.734} C_VEL
LIN {X 0,Y 198.424,Z 370.754,A -85,B 0,C 180,E1 -21907.787,E2 -21907.787} C_VEL
LIN {X 0,Y 194.719,Z 363.083,A -85,B 0,C 180,E1 -21909.309,E2 -21909.309} C_VEL
LIN {X 0,Y 193.269,Z 360.105,A -85,B 0,C 180,E1 -21909.887,E2 -21909.887} C_VEL
LIN {X 0,Y 193.06,Z 359.24,A -85,B 0,C 180,E1 -21910.031,E2 -21910.031} C_VEL
LIN {X 0,Y 192.765,Z 357.19,A -85,B 0,C 180,E1 -21913.846,E2 -21913.846} C_VEL
LIN {X 0,Y 192.525,Z 355.674,A -85,B 0,C 180,E1 -21916.894,E2 -21916.894} C_VEL
LIN {X 0,Y 192.541,Z 355.503,A -85,B 0,C 180,E1 -21921.646,E2 -21921.646} C_VEL
LIN {X 0,Y 192.595,Z 355.496,A -85,B 0,C 180,E1 -21926.813,E2 -21926.813} C_VEL
LIN {X 0,Y 192.62,Z 355.488,A -85,B 0,C 180,E1 -21931.685,E2 -21931.685} C_VEL
LIN {X 0,Y 192.679,Z 355.483,A -85,B 0,C 180,E1 -21936.345,E2 -21936.345} C_VEL
LIN {X 0,Y 192.732,Z 355.478,A -85,B 0,C 180,E1 -21941.458,E2 -21941.458} C_VEL
LIN {X 0,Y 192.764,Z 355.472,A -85,B 0,C 180,E1 -21945.214,E2 -21945.214} C_VEL
LIN {X 0,Y 192.982,Z 355.446,A -85,B 0,C 180,E1 -21949.508,E2 -21949.508} C_VEL
LIN {X 0,Y 193.062,Z 355.436,A -85,B 0,C 180,E1 -21951.627,E2 -21951.627} C_VEL
LIN {X 0,Y 193.262,Z 355.412,A -85,B 0,C 180,E1 -21957.916,E2 -21957.916} C_VEL
LIN {X 0,Y 193.432,Z 355.391,A -85,B 0,C 180,E1 -21960,E2 -21960} C_VEL
LIN {X 0,Y 192.971,Z 355.448,A -85,B 0,C 180,E1 -21964.177,E2 -21964.177} C_VEL
LIN {X 0,Y 193.036,Z 355.44,A -85,B 0,C 180,E1 -21968.374,E2 -21968.374} C_VEL
LIN {X 0,Y 192.802,Z 355.471,A -85,B 0,C 180,E1 -21972.633,E2 -21972.633} C_VEL
LIN {X 0,Y 192.757,Z 355.477,A -85,B 0,C 180,E1 -21976.959,E2 -21976.959} C_VEL
LIN {X 0,Y 192.62,Z 355.494,A -85,B 0,C 180,E1 -21981.399,E2 -21981.399} C_VEL
LIN {X 0,Y 192.639,Z 355.489,A -85,B 0,C 180,E1 -21984.208,E2 -21984.208} C_VEL
LIN {X 0,Y 192.602,Z 355.496,A -85,B 0,C 180,E1 -21988.866,E2 -21988.866} C_VEL
LIN {X 0,Y 192.68,Z 355.71,A -85,B 0,C 180,E1 -21991.862,E2 -21991.862} C_VEL
LIN {X 0,Y 193.102,Z 358.524,A -85,B 0,C 180,E1 -21996.803,E2 -21996.803} C_VEL
LIN {X 0,Y 193.481,Z 361.056,A -85,B 0,C 180,E1 -22000.831,E2 -22000.831} C_VEL
LIN {X 0,Y 193.82,Z 362.862,A -85,B 0,C 180,E1 -22003.547,E2 -22003.547} C_VEL
LIN {X 0,Y 194.373,Z 366.023,A -85,B 0,C 180,E1 -22008.018,E2 -22008.018} C_VEL
LIN {X 0,Y 194.627,Z 367.849,A -85,B 0,C 180,E1 -22010.418,E2 -22010.418} C_VEL
LIN {X 0,Y 195.645,Z 371.01,A -85,B 0,C 180,E1 -22010.87,E2 -22010.87} C_VEL
LIN {X 0,Y 196.882,Z 373.612,A -85,B 0,C 180,E1 -22011.345,E2 -22011.345} C_VEL
LIN {X 0,Y 200.191,Z 382.563,A -85,B 0,C 180,E1 -22012.877,E2 -22012.877} C_VEL
LIN {X 0,Y 202.84,Z 394.22,A -85,B 0,C 180,E1 -22014.786,E2 -22014.786} C_VEL
LIN {X 0,Y 204.296,Z 404.561,A -85,B 0,C 180,E1 -22016.604,E2 -22016.604} C_VEL
LIN {X 0,Y 205.023,Z 414.858,A -85,B 0,C 180,E1 -22018.608,E2 -22018.608} C_VEL
LIN {X 0,Y 204.843,Z 425.985,A -85,B 0,C 180,E1 -22021.043,E2 -22021.043} C_VEL
LIN {X 0,Y 204.345,Z 430.227,A -85,B 0,C 180,E1 -22022.056,E2 -22022.056} C_VEL
LIN {X 0,Y 201.611,Z 438.748,A -85,B 0,C 180,E1 -22024.167,E2 -22024.167} C_VEL
LIN {X 0,Y 198.599,Z 447.995,A -85,B 0,C 180,E1 -22027.091,E2 -22027.091} C_VEL
LIN {X 0,Y 195.898,Z 455.424,A -85,B 0,C 180,E1 -22030.073,E2 -22030.073} C_VEL
LIN {X 0,Y 193.777,Z 461.397,A -85,B 0,C 180,E1 -22033.133,E2 -22033.133} C_VEL
LIN {X 0,Y 192.164,Z 466.119,A -85,B 0,C 180,E1 -22036.247,E2 -22036.247} C_VEL
LIN {X 0,Y 191.041,Z 469.853,A -85,B 0,C 180,E1 -22039.539,E2 -22039.539} C_VEL
LIN {X 0,Y 189.966,Z 471.371,A -85,B 0,C 180,E1 -22041.236,E2 -22041.236} C_VEL
LIN {X 0,Y 186.707,Z 473.159,A -85,B 0,C 180,E1 -22044.033,E2 -22044.033} C_VEL
LIN {X 0,Y 184.172,Z 474.085,A -85,B 0,C 180,E1 -22046.354,E2 -22046.354} C_VEL
LIN {X 0,Y 183.144,Z 474.474,A -85,B 0,C 180,E1 -22048.178,E2 -22048.178} C_VEL
LIN {X 0,Y 183.081,Z 474.492,A -85,B 0,C 180,E1 -22048.797,E2 -22048.797} C_VEL
LIN {X 0,Y 183.163,Z 474.61,A -85,B 0,C 180,E1 -22049.999,E2 -22049.999} C_VEL
LIN {X 0,Y 183.053,Z 474.112,A -85,B 0,C 180,E1 -22053.413,E2 -22053.413} C_VEL
LIN {X 0,Y 183.229,Z 472.758,A -85,B 0,C 180,E1 -22056.607,E2 -22056.607} C_VEL
LIN {X 0,Y 183.55,Z 471.348,A -85,B 0,C 180,E1 -22058.809,E2 -22058.809} C_VEL
LIN {X 0,Y 184.403,Z 468.394,A -85,B 0,C 180,E1 -22062.099,E2 -22062.099} C_VEL
LIN {X 0,Y 185.688,Z 464.401,A -85,B 0,C 180,E1 -22065.362,E2 -22065.362} C_VEL
LIN {X 0,Y 188.071,Z 458.275,A -85,B 0,C 180,E1 -22069.084,E2 -22069.084} C_VEL
LIN {X 0,Y 190.615,Z 451.678,A -85,B 0,C 180,E1 -22072.161,E2 -22072.161} C_VEL
LIN {X 0,Y 193.459,Z 443.285,A -85,B 0,C 180,E1 -22075.266,E2 -22075.266} C_VEL
LIN {X 0,Y 196.401,Z 434.78,A -85,B 0,C 180,E1 -22077.721,E2 -22077.721} C_VEL
LIN {X 0,Y 197.956,Z 429.813,A -85,B 0,C 180,E1 -22078.927,E2 -22078.927} C_VEL
LIN {X 0,Y 198.51,Z 420.359,A -85,B 0,C 180,E1 -22081.229,E2 -22081.229} C_VEL
LIN {X 0,Y 198.272,Z 408.93,A -85,B 0,C 180,E1 -22083.664,E2 -22083.664} C_VEL
LIN {X 0,Y 197.03,Z 397.982,A -85,B 0,C 180,E1 -22085.772,E2 -22085.772} C_VEL
LIN {X 0,Y 194.693,Z 386.315,A -85,B 0,C 180,E1 -22087.853,E2 -22087.853} C_VEL
LIN {X 0,Y 191.401,Z 376.435,A -85,B 0,C 180,E1 -22089.645,E2 -22089.645} C_VEL
LIN {X 0,Y 189.135,Z 371.631,A -85,B 0,C 180,E1 -22090.611,E2 -22090.611} C_VEL
LIN {X 0,Y 187.604,Z 368.262,A -85,B 0,C 180,E1 -22091.261,E2 -22091.261} C_VEL
LIN {X 0,Y 187.46,Z 367.487,A -85,B 0,C 180,E1 -22091.426,E2 -22091.426} C_VEL
LIN {X 0,Y 186.911,Z 364.63,A -85,B 0,C 180,E1 -22095.593,E2 -22095.593} C_VEL
LIN {X 0,Y 186.399,Z 361.718,A -85,B 0,C 180,E1 -22100.136,E2 -22100.136} C_VEL
LIN {X 0,Y 186.144,Z 360.092,A -85,B 0,C 180,E1 -22102.836,E2 -22102.836} C_VEL
LIN {X 0,Y 185.743,Z 357.234,A -85,B 0,C 180,E1 -22108.013,E2 -22108.013} C_VEL
LIN {X 0,Y 185.511,Z 356.38,A -85,B 0,C 180,E1 -22109.87,E2 -22109.87} C_VEL
LIN {X 0,Y 185.575,Z 356.371,A -85,B 0,C 180,E1 -22115.381,E2 -22115.381} C_VEL
LIN {X 0,Y 185.669,Z 356.358,A -85,B 0,C 180,E1 -22121.133,E2 -22121.133} C_VEL
LIN {X 0,Y 185.758,Z 356.345,A -85,B 0,C 180,E1 -22126.879,E2 -22126.879} C_VEL
LIN {X 0,Y 186.003,Z 356.315,A -85,B 0,C 180,E1 -22131.307,E2 -22131.307} C_VEL
LIN {X 0,Y 186.202,Z 356.292,A -85,B 0,C 180,E1 -22137.837,E2 -22137.837} C_VEL
LIN {X 0,Y 186.391,Z 356.266,A -85,B 0,C 180,E1 -22140,E2 -22140} C_VEL
LIN {X 0,Y 185.92,Z 356.325,A -85,B 0,C 180,E1 -22144.336,E2 -22144.336} C_VEL
LIN {X 0,Y 186.023,Z 356.31,A -85,B 0,C 180,E1 -22148.692,E2 -22148.692} C_VEL
LIN {X 0,Y 185.729,Z 356.351,A -85,B 0,C 180,E1 -22153.123,E2 -22153.123} C_VEL
LIN {X 0,Y 185.685,Z 356.355,A -85,B 0,C 180,E1 -22157.626,E2 -22157.626} C_VEL
LIN {X 0,Y 185.572,Z 356.367,A -85,B 0,C 180,E1 -22162.255,E2 -22162.255} C_VEL
LIN {X 0,Y 185.503,Z 356.378,A -85,B 0,C 180,E1 -22167.042,E2 -22167.042} C_VEL
LIN {X 0,Y 185.539,Z 356.374,A -85,B 0,C 180,E1 -22169.5,E2 -22169.5} C_VEL
LIN {X 0,Y 185.493,Z 356.379,A -85,B 0,C 180,E1 -22174.634,E2 -22174.634} C_VEL
LIN {X 0,Y 185.496,Z 356.379,A -85,B 0,C 180,E1 -22177.316,E2 -22177.316} C_VEL
LIN {X 0,Y 185.458,Z 356.381,A -85,B 0,C 180,E1 -22180.723,E2 -22180.723} C_VEL
LIN {X 0,Y 185.625,Z 357.39,A -85,B 0,C 180,E1 -22184.001,E2 -22184.001} C_VEL
LIN {X 0,Y 185.937,Z 359.557,A -85,B 0,C 180,E1 -22188.323,E2 -22188.323} C_VEL
LIN {X 0,Y 187.134,Z 362.587,A -85,B 0,C 180,E1 -22188.878,E2 -22188.878} C_VEL
LIN {X 0,Y 188.611,Z 364.832,A -85,B 0,C 180,E1 -22189.448,E2 -22189.448} C_VEL
LIN {X 0,Y 193.437,Z 375.364,A -85,B 0,C 180,E1 -22191.712,E2 -22191.712} C_VEL
LIN {X 0,Y 196.741,Z 385.428,A -85,B 0,C 180,E1 -22193.785,E2 -22193.785} C_VEL
LIN {X 0,Y 199.099,Z 396.272,A -85,B 0,C 180,E1 -22196.049,E2 -22196.049} C_VEL
LIN {X 0,Y 200.352,Z 406.111,A -85,B 0,C 180,E1 -22198.254,E2 -22198.254} C_VEL
LIN {X 0,Y 200.719,Z 413.558,A -85,B 0,C 180,E1 -22200.071,E2 -22200.071} C_VEL
LIN {X 0,Y 197.684,Z 424.024,A -85,B 0,C 180,E1 -22202.474,E2 -22202.474} C_VEL
LIN {X 0,Y 194.949,Z 432.49,A -85,B 0,C 180,E1 -22204.94,E2 -22204.94} C_VEL
LIN {X 0,Y 191.84,Z 440.73,A -85,B 0,C 180,E1 -22207.946,E2 -22207.946} C_VEL
LIN {X 0,Y 189.535,Z 446.366,A -85,B 0,C 180,E1 -22210.507,E2 -22210.507} C_VEL
LIN {X 0,Y 187.39,Z 451.853,A -85,B 0,C 180,E1 -22213.664,E2 -22213.664} C_VEL
LIN {X 0,Y 185.658,Z 456.159,A -85,B 0,C 180,E1 -22216.873,E2 -22216.873} C_VEL
LIN {X 0,Y 184.784,Z 458.436,A -85,B 0,C 180,E1 -22219.039,E2 -22219.039} C_VEL
LIN {X 0,Y 184.168,Z 460.284,A -85,B 0,C 180,E1 -22221.221,E2 -22221.221} C_VEL
LIN {X 0,Y 183.497,Z 462.347,A -85,B 0,C 180,E1 -22224.756,E2 -22224.756} C_VEL
LIN {X 0,Y 183.248,Z 463.264,A -85,B 0,C 180,E1 -22227.803,E2 -22227.803} C_VEL
LIN {X 0,Y 183.233,Z 463.49,A -85,B 0,C 180,E1 -22230.001,E2 -22230.001} C_VEL
LIN {X 0,Y 183.246,Z 463.295,A -85,B 0,C 180,E1 -22232.199,E2 -22232.199} C_VEL
LIN {X 0,Y 183.694,Z 461.742,A -85,B 0,C 180,E1 -22236.592,E2 -22236.592} C_VEL
LIN {X 0,Y 184.173,Z 460.385,A -85,B 0,C 180,E1 -22238.781,E2 -22238.781} C_VEL
LIN {X 0,Y 185.199,Z 457.518,A -85,B 0,C 180,E1 -22242.048,E2 -22242.048} C_VEL
LIN {X 0,Y 186.727,Z 453.627,A -85,B 0,C 180,E1 -22245.276,E2 -22245.276} C_VEL
LIN {X 0,Y 188.72,Z 448.606,A -85,B 0,C 180,E1 -22248.455,E2 -22248.455} C_VEL
LIN {X 0,Y 191.263,Z 442.277,A -85,B 0,C 180,E1 -22251.559,E2 -22251.559} C_VEL
LIN {X 0,Y 194.294,Z 434.357,A -85,B 0,C 180,E1 -22254.581,E2 -22254.581} C_VEL
LIN {X 0,Y 196.962,Z 426.334,A -85,B 0,C 180,E1 -22257.047,E2 -22257.047} C_VEL
LIN {X 0,Y 200.131,Z 416.434,A -85,B 0,C 180,E1 -22259.449,E2 -22259.449} C_VEL
LIN {X 0,Y 200.75,Z 414.163,A -85,B 0,C 180,E1 -22259.926,E2 -22259.926} C_VEL
LIN {X 0,Y 200.23,Z 404.34,A -85,B 0,C 180,E1 -22262.296,E2 -22262.296} C_VEL
LIN {X 0,Y 198.669,Z 393.598,A -85,B 0,C 180,E1 -22264.666,E2 -22264.666} C_VEL
LIN {X 0,Y 196.106,Z 383.218,A -85,B 0,C 180,E1 -22266.835,E2 -22266.835} C_VEL
LIN {X 0,Y 192.532,Z 373.122,A -85,B 0,C 180,E1 -22268.923,E2 -22268.923} C_VEL
LIN {X 0,Y 188.031,Z 363.831,A -85,B 0,C 180,E1 -22270.959,E2 -22270.959} C_VEL
LIN {X 0,Y 186.212,Z 360.692,A -85,B 0,C 180,E1 -22271.702,E2 -22271.702} C_VEL
LIN {X 0,Y 185.903,Z 359.514,A -85,B 0,C 180,E1 -22271.879,E2 -22271.879} C_VEL
LIN {X 0,Y 185.608,Z 357.465,A -85,B 0,C 180,E1 -22276.008,E2 -22276.008} C_VEL
LIN {X 0,Y 185.462,Z 356.384,A -85,B 0,C 180,E1 -22279.279,E2 -22279.279} C_VEL
LIN {X 0,Y 185.501,Z 356.376,A -85,B 0,C 180,E1 -22282.714,E2 -22282.714} C_VEL
LIN {X 0,Y 185.531,Z 356.37,A -85,B 0,C 180,E1 -22287.972,E2 -22287.972} C_VEL
LIN {X 0,Y 185.547,Z 356.37,A -85,B 0,C 180,E1 -22290.595,E2 -22290.595} C_VEL
LIN {X 0,Y 185.581,Z 356.363,A -85,B 0,C 180,E1 -22295.381,E2 -22295.381} C_VEL
LIN {X 0,Y 185.675,Z 356.357,A -85,B 0,C 180,E1 -22301.134,E2 -22301.134} C_VEL
LIN {X 0,Y 185.695,Z 356.354,A -85,B 0,C 180,E1 -22304.637,E2 -22304.637} C_VEL
LIN {X 0,Y 185.925,Z 356.325,A -85,B 0,C 180,E1 -22309.359,E2 -22309.359} C_VEL
LIN {X 0,Y 185.961,Z 356.319,A -85,B 0,C 180,E1 -22313.49,E2 -22313.49} C_VEL
LIN {X 0,Y 186.206,Z 356.291,A -85,B 0,C 180,E1 -22317.837,E2 -22317.837} C_VEL
LIN {X 0,Y 186.397,Z 356.267,A -85,B 0,C 180,E1 -22320,E2 -22320} C_VEL
LIN {X 0,Y 185.918,Z 356.327,A -85,B 0,C 180,E1 -22324.336,E2 -22324.336} C_VEL
LIN {X 0,Y 185.983,Z 356.319,A -85,B 0,C 180,E1 -22328.694,E2 -22328.694} C_VEL
LIN {X 0,Y 185.729,Z 356.352,A -85,B 0,C 180,E1 -22333.123,E2 -22333.123} C_VEL
LIN {X 0,Y 185.69,Z 356.357,A -85,B 0,C 180,E1 -22337.625,E2 -22337.625} C_VEL
LIN {X 0,Y 185.578,Z 356.368,A -85,B 0,C 180,E1 -22342.254,E2 -22342.254} C_VEL
LIN {X 0,Y 185.508,Z 356.379,A -85,B 0,C 180,E1 -22347.041,E2 -22347.041} C_VEL
LIN {X 0,Y 185.554,Z 356.522,A -85,B 0,C 180,E1 -22350.437,E2 -22350.437} C_VEL
LIN {X 0,Y 185.935,Z 358.656,A -85,B 0,C 180,E1 -22354.539,E2 -22354.539} C_VEL
LIN {X 0,Y 186.405,Z 361.774,A -85,B 0,C 180,E1 -22359.863,E2 -22359.863} C_VEL
LIN {X 0,Y 186.877,Z 364.681,A -85,B 0,C 180,E1 -22364.394,E2 -22364.394} C_VEL
LIN {X 0,Y 187.436,Z 367.71,A -85,B 0,C 180,E1 -22368.583,E2 -22368.583} C_VEL
LIN {X 0,Y 188.629,Z 370.886,A -85,B 0,C 180,E1 -22369.124,E2 -22369.124} C_VEL
LIN {X 0,Y 189.896,Z 373.108,A -85,B 0,C 180,E1 -22369.619,E2 -22369.619} C_VEL
LIN {X 0,Y 193.257,Z 381.578,A -85,B 0,C 180,E1 -22371.225,E2 -22371.225} C_VEL
LIN {X 0,Y 195.401,Z 389.228,A -85,B 0,C 180,E1 -22372.597,E2 -22372.597} C_VEL
LIN {X 0,Y 197.476,Z 400.624,A -85,B 0,C 180,E1 -22374.667,E2 -22374.667} C_VEL
LIN {X 0,Y 198.47,Z 411.843,A -85,B 0,C 180,E1 -22376.868,E2 -22376.868} C_VEL
LIN {X 0,Y 198.549,Z 421.806,A -85,B 0,C 180,E1 -22379.054,E2 -22379.054} C_VEL
LIN {X 0,Y 198.034,Z 430.012,A -85,B 0,C 180,E1 -22381.083,E2 -22381.083} C_VEL
LIN {X 0,Y 195.215,Z 438.535,A -85,B 0,C 180,E1 -22383.255,E2 -22383.255} C_VEL
LIN {X 0,Y 192.276,Z 447.169,A -85,B 0,C 180,E1 -22386.035,E2 -22386.035} C_VEL
LIN {X 0,Y 189.205,Z 455.21,A -85,B 0,C 180,E1 -22389.336,E2 -22389.336} C_VEL
LIN {X 0,Y 186.954,Z 461.181,A -85,B 0,C 180,E1 -22392.497,E2 -22392.497} C_VEL
LIN {X 0,Y 185.227,Z 465.903,A -85,B 0,C 180,E1 -22395.721,E2 -22395.721} C_VEL
LIN {X 0,Y 183.98,Z 469.822,A -85,B 0,C 180,E1 -22399.354,E2 -22399.354} C_VEL
LIN {X 0,Y 183.552,Z 471.38,A -85,B 0,C 180,E1 -22401.189,E2 -22401.189} C_VEL
LIN {X 0,Y 183.23,Z 472.78,A -85,B 0,C 180,E1 -22403.392,E2 -22403.392} C_VEL
LIN {X 0,Y 183.04,Z 474.138,A -85,B 0,C 180,E1 -22406.658,E2 -22406.658} C_VEL
LIN {X 0,Y 183.081,Z 474.492,A -85,B 0,C 180,E1 -22408.797,E2 -22408.797} C_VEL
LIN {X 0,Y 182.437,Z 474.559,A -85,B 0,C 180,E1 -22410.632,E2 -22410.632} C_VEL
LIN {X 0,Y 180.841,Z 474.293,A -85,B 0,C 180,E1 -22412.436,E2 -22412.436} C_VEL
LIN {X 0,Y 177.206,Z 472.952,A -85,B 0,C 180,E1 -22416.078,E2 -22416.078} C_VEL
LIN {X 0,Y 176.371,Z 471.905,A -85,B 0,C 180,E1 -22417.97,E2 -22417.97} C_VEL
LIN {X 0,Y 176.396,Z 471.475,A -85,B 0,C 180,E1 -22418.606,E2 -22418.606} C_VEL
LIN {X 0,Y 177.449,Z 468.177,A -85,B 0,C 180,E1 -22422.58,E2 -22422.58} C_VEL
LIN {X 0,Y 178.814,Z 464.183,A -85,B 0,C 180,E1 -22425.968,E2 -22425.968} C_VEL
LIN {X 0,Y 181.349,Z 458.057,A -85,B 0,C 180,E1 -22429.82,E2 -22429.82} C_VEL
LIN {X 0,Y 184.022,Z 451.493,A -85,B 0,C 180,E1 -22432.984,E2 -22432.984} C_VEL
LIN {X 0,Y 187.025,Z 443.065,A -85,B 0,C 180,E1 -22436.201,E2 -22436.201} C_VEL
LIN {X 0,Y 190.118,Z 434.56,A -85,B 0,C 180,E1 -22438.721,E2 -22438.721} C_VEL
LIN {X 0,Y 191.535,Z 429.585,A -85,B 0,C 180,E1 -22439.994,E2 -22439.994} C_VEL
LIN {X 0,Y 192.118,Z 420.127,A -85,B 0,C 180,E1 -22442.392,E2 -22442.392} C_VEL
LIN {X 0,Y 191.933,Z 409.624,A -85,B 0,C 180,E1 -22444.748,E2 -22444.748} C_VEL
LIN {X 0,Y 190.802,Z 398.744,A -85,B 0,C 180,E1 -22446.966,E2 -22446.966} C_VEL
LIN {X 0,Y 188.673,Z 387.68,A -85,B 0,C 180,E1 -22449.077,E2 -22449.077} C_VEL
LIN {X 0,Y 185.645,Z 379.02,A -85,B 0,C 180,E1 -22450.857,E2 -22450.857} C_VEL
LIN {X 0,Y 184.153,Z 375.713,A -85,B 0,C 180,E1 -22451.581,E2 -22451.581} C_VEL
LIN {X 0,Y 182.357,Z 371.89,A -85,B 0,C 180,E1 -22452.418,E2 -22452.418} C_VEL
LIN {X 0,Y 180.579,Z 368.812,A -85,B 0,C 180,E1 -22453.185,E2 -22453.185} C_VEL
LIN {X 0,Y 180.153,Z 367.239,A -85,B 0,C 180,E1 -22453.472,E2 -22453.472} C_VEL
LIN {X 0,Y 179.587,Z 364.166,A -85,B 0,C 180,E1 -22458.296,E2 -22458.296} C_VEL
LIN {X 0,Y 179.256,Z 362.183,A -85,B 0,C 180,E1 -22461.637,E2 -22461.637} C_VEL
LIN {X 0,Y 178.868,Z 359.441,A -85,B 0,C 180,E1 -22466.627,E2 -22466.627} C_VEL
LIN {X 0,Y 178.465,Z 357.257,A -85,B 0,C 180,E1 -22471.341,E2 -22471.341} C_VEL
LIN {X 0,Y 178.51,Z 357.251,A -85,B 0,C 180,E1 -22474.888,E2 -22474.888} C_VEL
LIN {X 0,Y 178.617,Z 357.237,A -85,B 0,C 180,E1 -22480.785,E2 -22480.785} C_VEL
LIN {X 0,Y 178.675,Z 357.228,A -85,B 0,C 180,E1 -22486.349,E2 -22486.349} C_VEL
LIN {X 0,Y 178.954,Z 357.193,A -85,B 0,C 180,E1 -22490.962,E2 -22490.962} C_VEL
LIN {X 0,Y 179.148,Z 357.169,A -85,B 0,C 180,E1 -22497.752,E2 -22497.752} C_VEL
LIN {X 0,Y 179.356,Z 357.142,A -85,B 0,C 180,E1 -22500,E2 -22500} C_VEL
LIN {X 0,Y 178.869,Z 357.204,A -85,B 0,C 180,E1 -22504.507,E2 -22504.507} C_VEL
LIN {X 0,Y 178.972,Z 357.189,A -85,B 0,C 180,E1 -22509.037,E2 -22509.037} C_VEL
LIN {X 0,Y 178.656,Z 357.229,A -85,B 0,C 180,E1 -22513.652,E2 -22513.652} C_VEL
LIN {X 0,Y 178.617,Z 357.235,A -85,B 0,C 180,E1 -22519.216,E2 -22519.216} C_VEL
LIN {X 0,Y 178.51,Z 357.249,A -85,B 0,C 180,E1 -22525.112,E2 -22525.112} C_VEL
LIN {X 0,Y 178.455,Z 357.256,A -85,B 0,C 180,E1 -22530.795,E2 -22530.795} C_VEL
LIN {X 0,Y 178.478,Z 357.253,A -85,B 0,C 180,E1 -22534.219,E2 -22534.219} C_VEL
LIN {X 0,Y 178.384,Z 357.265,A -85,B 0,C 180,E1 -22539.078,E2 -22539.078} C_VEL
LIN {X 0,Y 178.482,Z 357.878,A -85,B 0,C 180,E1 -22542.021,E2 -22542.021} C_VEL
LIN {X 0,Y 178.859,Z 359.902,A -85,B 0,C 180,E1 -22546.273,E2 -22546.273} C_VEL
LIN {X 0,Y 179.997,Z 362.83,A -85,B 0,C 180,E1 -22546.858,E2 -22546.858} C_VEL
LIN {X 0,Y 181.733,Z 365.494,A -85,B 0,C 180,E1 -22547.596,E2 -22547.596} C_VEL
LIN {X 0,Y 184.884,Z 371.575,A -85,B 0,C 180,E1 -22549.097,E2 -22549.097} C_VEL
LIN {X 0,Y 188.914,Z 381.375,A -85,B 0,C 180,E1 -22551.375,E2 -22551.375} C_VEL
LIN {X 0,Y 191.787,Z 391.988,A -85,B 0,C 180,E1 -22553.725,E2 -22553.725} C_VEL
LIN {X 0,Y 193.464,Z 402.027,A -85,B 0,C 180,E1 -22556.025,E2 -22556.025} C_VEL
LIN {X 0,Y 194.206,Z 411.693,A -85,B 0,C 180,E1 -22558.409,E2 -22558.409} C_VEL
LIN {X 0,Y 194.292,Z 415,A -85,B 0,C 180,E1 -22559.29,E2 -22559.29} C_VEL
LIN {X 0,Y 191.403,Z 424.243,A -85,B 0,C 180,E1 -22561.49,E2 -22561.49} C_VEL
LIN {X 0,Y 188.538,Z 432.708,A -85,B 0,C 180,E1 -22564.025,E2 -22564.025} C_VEL
LIN {X 0,Y 185.281,Z 440.947,A -85,B 0,C 180,E1 -22567.122,E2 -22567.122} C_VEL
LIN {X 0,Y 182.856,Z 446.583,A -85,B 0,C 180,E1 -22569.764,E2 -22569.764} C_VEL
LIN {X 0,Y 180.576,Z 452.071,A -85,B 0,C 180,E1 -22573.03,E2 -22573.03} C_VEL
LIN {X 0,Y 178.744,Z 456.376,A -85,B 0,C 180,E1 -22576.356,E2 -22576.356} C_VEL
LIN {X 0,Y 177.821,Z 458.653,A -85,B 0,C 180,E1 -22578.604,E2 -22578.604} C_VEL
LIN {X 0,Y 177.163,Z 460.5,A -85,B 0,C 180,E1 -22580.871,E2 -22580.871} C_VEL
LIN {X 0,Y 176.395,Z 462.697,A -85,B 0,C 180,E1 -22584.916,E2 -22584.916} C_VEL
LIN {X 0,Y 176.162,Z 463.48,A -85,B 0,C 180,E1 -22587.715,E2 -22587.715} C_VEL
LIN {X 0,Y 176.141,Z 463.705,A -85,B 0,C 180,E1 -22590.001,E2 -22590.001} C_VEL
LIN {X 0,Y 176.16,Z 463.51,A -85,B 0,C 180,E1 -22592.287,E2 -22592.287} C_VEL
LIN {X 0,Y 176.364,Z 462.787,A -85,B 0,C 180,E1 -22594.971,E2 -22594.971} C_VEL
LIN {X 0,Y 177.169,Z 460.6,A -85,B 0,C 180,E1 -22599.131,E2 -22599.131} C_VEL
LIN {X 0,Y 178.244,Z 457.733,A -85,B 0,C 180,E1 -22602.525,E2 -22602.525} C_VEL
LIN {X 0,Y 179.867,Z 453.842,A -85,B 0,C 180,E1 -22605.874,E2 -22605.874} C_VEL
LIN {X 0,Y 181.975,Z 448.82,A -85,B 0,C 180,E1 -22609.165,E2 -22609.165} C_VEL
LIN {X 0,Y 184.681,Z 442.49,A -85,B 0,C 180,E1 -22612.368,E2 -22612.368} C_VEL
LIN {X 0,Y 187.846,Z 434.571,A -85,B 0,C 180,E1 -22615.484,E2 -22615.484} C_VEL
LIN {X 0,Y 190.941,Z 425.761,A -85,B 0,C 180,E1 -22618.238,E2 -22618.238} C_VEL
LIN {X 0,Y 194.292,Z 415.569,A -85,B 0,C 180,E1 -22620.72,E2 -22620.72} C_VEL
LIN {X 0,Y 193.922,Z 405.875,A -85,B 0,C 180,E1 -22623.193,E2 -22623.193} C_VEL
LIN {X 0,Y 192.73,Z 396.562,A -85,B 0,C 180,E1 -22625.39,E2 -22625.39} C_VEL
LIN {X 0,Y 190.205,Z 385.584,A -85,B 0,C 180,E1 -22627.857,E2 -22627.857} C_VEL
LIN {X 0,Y 187.387,Z 377.186,A -85,B 0,C 180,E1 -22629.746,E2 -22629.746} C_VEL
LIN {X 0,Y 183.317,Z 368.45,A -85,B 0,C 180,E1 -22631.838,E2 -22631.838} C_VEL
LIN {X 0,Y 180.802,Z 363.959,A -85,B 0,C 180,E1 -22632.991,E2 -22632.991} C_VEL
LIN {X 0,Y 179.112,Z 360.936,A -85,B 0,C 180,E1 -22633.761,E2 -22633.761} C_VEL
LIN {X 0,Y 178.829,Z 359.787,A -85,B 0,C 180,E1 -22633.971,E2 -22633.971} C_VEL
LIN {X 0,Y 178.479,Z 357.773,A -85,B 0,C 180,E1 -22638.432,E2 -22638.432} C_VEL
LIN {X 0,Y 178.407,Z 357.262,A -85,B 0,C 180,E1 -22641.986,E2 -22641.986} C_VEL
LIN {X 0,Y 178.484,Z 357.253,A -85,B 0,C 180,E1 -22646.546,E2 -22646.546} C_VEL
LIN {X 0,Y 178.444,Z 357.253,A -85,B 0,C 180,E1 -22651.795,E2 -22651.795} C_VEL
LIN {X 0,Y 178.516,Z 357.242,A -85,B 0,C 180,E1 -22654.889,E2 -22654.889} C_VEL
LIN {X 0,Y 178.623,Z 357.234,A -85,B 0,C 180,E1 -22660.785,E2 -22660.785} C_VEL
LIN {X 0,Y 178.661,Z 357.23,A -85,B 0,C 180,E1 -22666.348,E2 -22666.348} C_VEL
LIN {X 0,Y 178.96,Z 357.192,A -85,B 0,C 180,E1 -22670.962,E2 -22670.962} C_VEL
LIN {X 0,Y 179.152,Z 357.169,A -85,B 0,C 180,E1 -22677.752,E2 -22677.752} C_VEL
LIN {X 0,Y 179.361,Z 357.144,A -85,B 0,C 180,E1 -22680,E2 -22680} C_VEL
LIN {X 0,Y 178.866,Z 357.206,A -85,B 0,C 180,E1 -22684.507,E2 -22684.507} C_VEL
LIN {X 0,Y 178.911,Z 357.2,A -85,B 0,C 180,E1 -22689.04,E2 -22689.04} C_VEL
LIN {X 0,Y 178.657,Z 357.232,A -85,B 0,C 180,E1 -22693.652,E2 -22693.652} C_VEL
LIN {X 0,Y 178.623,Z 357.238,A -85,B 0,C 180,E1 -22699.215,E2 -22699.215} C_VEL
LIN {X 0,Y 178.516,Z 357.25,A -85,B 0,C 180,E1 -22705.111,E2 -22705.111} C_VEL
LIN {X 0,Y 178.444,Z 357.259,A -85,B 0,C 180,E1 -22708.204,E2 -22708.204} C_VEL
LIN {X 0,Y 178.66,Z 358.202,A -85,B 0,C 180,E1 -22710.756,E2 -22710.756} C_VEL
LIN {X 0,Y 178.996,Z 360.061,A -85,B 0,C 180,E1 -22714.459,E2 -22714.459} C_VEL
LIN {X 0,Y 179.302,Z 362.516,A -85,B 0,C 180,E1 -22718.84,E2 -22718.84} C_VEL
LIN {X 0,Y 179.632,Z 364.389,A -85,B 0,C 180,E1 -22721.981,E2 -22721.981} C_VEL
LIN {X 0,Y 180.17,Z 367.483,A -85,B 0,C 180,E1 -22726.514,E2 -22726.514} C_VEL
LIN {X 0,Y 181.316,Z 370.482,A -85,B 0,C 180,E1 -22727.082,E2 -22727.082} C_VEL
LIN {X 0,Y 182.901,Z 372.983,A -85,B 0,C 180,E1 -22727.74,E2 -22727.74} C_VEL
LIN {X 0,Y 186.519,Z 381.154,A -85,B 0,C 180,E1 -22729.523,E2 -22729.523} C_VEL
LIN {X 0,Y 189.221,Z 389.816,A -85,B 0,C 180,E1 -22731.259,E2 -22731.259} C_VEL
LIN {X 0,Y 191.055,Z 399.891,A -85,B 0,C 180,E1 -22733.209,E2 -22733.209} C_VEL
LIN {X 0,Y 192.042,Z 410.995,A -85,B 0,C 180,E1 -22735.483,E2 -22735.483} C_VEL
LIN {X 0,Y 192.163,Z 421.414,A -85,B 0,C 180,E1 -22737.863,E2 -22737.863} C_VEL
LIN {X 0,Y 191.475,Z 430.836,A -85,B 0,C 180,E1 -22740.296,E2 -22740.296} C_VEL
LIN {X 0,Y 188.273,Z 439.993,A -85,B 0,C 180,E1 -22742.788,E2 -22742.788} C_VEL
LIN {X 0,Y 184.912,Z 449.169,A -85,B 0,C 180,E1 -22745.991,E2 -22745.991} C_VEL
LIN {X 0,Y 182.121,Z 456.111,A -85,B 0,C 180,E1 -22749.086,E2 -22749.086} C_VEL
LIN {X 0,Y 180.165,Z 460.966,A -85,B 0,C 180,E1 -22751.815,E2 -22751.815} C_VEL
LIN {X 0,Y 178.317,Z 465.687,A -85,B 0,C 180,E1 -22755.155,E2 -22755.155} C_VEL
LIN {X 0,Y 177.081,Z 469.3,A -85,B 0,C 180,E1 -22758.553,E2 -22758.553} C_VEL
LIN {X 0,Y 176.51,Z 471.164,A -85,B 0,C 180,E1 -22760.835,E2 -22760.835} C_VEL
LIN {X 0,Y 176.009,Z 473.566,A -85,B 0,C 180,E1 -22765.419,E2 -22765.419} C_VEL
LIN {X 0,Y 175.985,Z 474.284,A -85,B 0,C 180,E1 -22768.83,E2 -22768.83} C_VEL
LIN {X 0,Y 176.071,Z 474.395,A -85,B 0,C 180,E1 -22769.999,E2 -22769.999} C_VEL
LIN {X 0,Y 175.97,Z 473.978,A -85,B 0,C 180,E1 -22773.174,E2 -22773.174} C_VEL
LIN {X 0,Y 176.155,Z 472.541,A -85,B 0,C 180,E1 -22776.873,E2 -22776.873} C_VEL
LIN {X 0,Y 176.396,Z 471.475,A -85,B 0,C 180,E1 -22778.606,E2 -22778.606} C_VEL
LIN {X 0,Y 176.134,Z 470.168,A -85,B 0,C 180,E1 -22780.477,E2 -22780.477} C_VEL
LIN {X 0,Y 174.194,Z 467.427,A -85,B 0,C 180,E1 -22783.532,E2 -22783.532} C_VEL
LIN {X 0,Y 172.659,Z 463.967,A -85,B 0,C 180,E1 -22786.57,E2 -22786.57} C_VEL
LIN {X 0,Y 173.035,Z 461.505,A -85,B 0,C 180,E1 -22788.354,E2 -22788.354} C_VEL
LIN {X 0,Y 175.469,Z 455.794,A -85,B 0,C 180,E1 -22791.744,E2 -22791.744} C_VEL
LIN {X 0,Y 178.142,Z 449.539,A -85,B 0,C 180,E1 -22794.651,E2 -22794.651} C_VEL
LIN {X 0,Y 181.279,Z 441.253,A -85,B 0,C 180,E1 -22797.723,E2 -22797.723} C_VEL
LIN {X 0,Y 184.61,Z 432.388,A -85,B 0,C 180,E1 -22800.291,E2 -22800.291} C_VEL
LIN {X 0,Y 185.545,Z 424.884,A -85,B 0,C 180,E1 -22802.362,E2 -22802.362} C_VEL
LIN {X 0,Y 185.83,Z 414.252,A -85,B 0,C 180,E1 -22804.992,E2 -22804.992} C_VEL
LIN {X 0,Y 185.136,Z 403.499,A -85,B 0,C 180,E1 -22807.398,E2 -22807.398} C_VEL
LIN {X 0,Y 183.46,Z 392.506,A -85,B 0,C 180,E1 -22809.686,E2 -22809.686} C_VEL
LIN {X 0,Y 180.784,Z 383.553,A -85,B 0,C 180,E1 -22811.642,E2 -22811.642} C_VEL
LIN {X 0,Y 177.581,Z 376.362,A -85,B 0,C 180,E1 -22813.392,E2 -22813.392} C_VEL
LIN {X 0,Y 175.213,Z 371.831,A -85,B 0,C 180,E1 -22814.568,E2 -22814.568} C_VEL
LIN {X 0,Y 173.399,Z 368.677,A -85,B 0,C 180,E1 -22815.437,E2 -22815.437} C_VEL
LIN {X 0,Y 172.895,Z 366.95,A -85,B 0,C 180,E1 -22815.782,E2 -22815.782} C_VEL
LIN {X 0,Y 172.362,Z 364.01,A -85,B 0,C 180,E1 -22820.777,E2 -22820.777} C_VEL
LIN {X 0,Y 172.014,Z 361.689,A -85,B 0,C 180,E1 -22825.11,E2 -22825.11} C_VEL
LIN {X 0,Y 171.592,Z 359.069,A -85,B 0,C 180,E1 -22830.561,E2 -22830.561} C_VEL
LIN {X 0,Y 171.384,Z 358.139,A -85,B 0,C 180,E1 -22833.187,E2 -22833.187} C_VEL
LIN {X 0,Y 171.446,Z 358.129,A -85,B 0,C 180,E1 -22838.35,E2 -22838.35} C_VEL
LIN {X 0,Y 171.573,Z 358.114,A -85,B 0,C 180,E1 -22840.871,E2 -22840.871} C_VEL
LIN {X 0,Y 171.588,Z 358.113,A -85,B 0,C 180,E1 -22845.774,E2 -22845.774} C_VEL
LIN {X 0,Y 171.883,Z 358.075,A -85,B 0,C 180,E1 -22850.587,E2 -22850.587} C_VEL
LIN {X 0,Y 171.818,Z 358.083,A -85,B 0,C 180,E1 -22855.308,E2 -22855.308} C_VEL
LIN {X 0,Y 172.32,Z 358.019,A -85,B 0,C 180,E1 -22860,E2 -22860} C_VEL
LIN {X 0,Y 171.818,Z 358.082,A -85,B 0,C 180,E1 -22864.693,E2 -22864.693} C_VEL
LIN {X 0,Y 171.898,Z 358.072,A -85,B 0,C 180,E1 -22869.413,E2 -22869.413} C_VEL
LIN {X 0,Y 171.573,Z 358.11,A -85,B 0,C 180,E1 -22874.228,E2 -22874.228} C_VEL
LIN {X 0,Y 171.536,Z 358.116,A -85,B 0,C 180,E1 -22879.559,E2 -22879.559} C_VEL
LIN {X 0,Y 171.439,Z 358.13,A -85,B 0,C 180,E1 -22885.599,E2 -22885.599} C_VEL
LIN {X 0,Y 171.413,Z 358.133,A -85,B 0,C 180,E1 -22890.574,E2 -22890.574} C_VEL
LIN {X 0,Y 171.388,Z 358.137,A -85,B 0,C 180,E1 -22895.036,E2 -22895.036} C_VEL
LIN {X 0,Y 171.34,Z 358.143,A -85,B 0,C 180,E1 -22898.803,E2 -22898.803} C_VEL
LIN {X 0,Y 171.635,Z 360.093,A -85,B 0,C 180,E1 -22903.873,E2 -22903.873} C_VEL
LIN {X 0,Y 173.051,Z 363.41,A -85,B 0,C 180,E1 -22904.687,E2 -22904.687} C_VEL
LIN {X 0,Y 174.625,Z 365.461,A -85,B 0,C 180,E1 -22905.397,E2 -22905.397} C_VEL
LIN {X 0,Y 176.669,Z 369.229,A -85,B 0,C 180,E1 -22906.449,E2 -22906.449} C_VEL
LIN {X 0,Y 180.562,Z 377.177,A -85,B 0,C 180,E1 -22908.573,E2 -22908.573} C_VEL
LIN {X 0,Y 184.079,Z 386.911,A -85,B 0,C 180,E1 -22910.996,E2 -22910.996} C_VEL
LIN {X 0,Y 186.237,Z 396.609,A -85,B 0,C 180,E1 -22913.311,E2 -22913.311} C_VEL
LIN {X 0,Y 187.533,Z 406.586,A -85,B 0,C 180,E1 -22915.798,E2 -22915.798} C_VEL
LIN {X 0,Y 187.864,Z 416.316,A -85,B 0,C 180,E1 -22918.418,E2 -22918.418} C_VEL
LIN {X 0,Y 184.559,Z 426.3,A -85,B 0,C 180,E1 -22920.969,E2 -22920.969} C_VEL
LIN {X 0,Y 181.035,Z 435.882,A -85,B 0,C 180,E1 -22924.106,E2 -22924.106} C_VEL
LIN {X 0,Y 177.682,Z 443.556,A -85,B 0,C 180,E1 -22927.318,E2 -22927.318} C_VEL
LIN {X 0,Y 175.353,Z 448.795,A -85,B 0,C 180,E1 -22930.084,E2 -22930.084} C_VEL
LIN {X 0,Y 173.097,Z 453.871,A -85,B 0,C 180,E1 -22933.49,E2 -22933.49} C_VEL
LIN {X 0,Y 171.329,Z 457.811,A -85,B 0,C 180,E1 -22936.962,E2 -22936.962} C_VEL
LIN {X 0,Y 170.149,Z 460.717,A -85,B 0,C 180,E1 -22940.491,E2 -22940.491} C_VEL
LIN {X 0,Y 169.659,Z 462.102,A -85,B 0,C 180,E1 -22942.862,E2 -22942.862} C_VEL
LIN {X 0,Y 169.079,Z 463.695,A -85,B 0,C 180,E1 -22947.619,E2 -22947.619} C_VEL
LIN {X 0,Y 169.052,Z 463.92,A -85,B 0,C 180,E1 -22950.001,E2 -22950.001} C_VEL
LIN {X 0,Y 169.077,Z 463.725,A -85,B 0,C 180,E1 -22952.383,E2 -22952.383} C_VEL
LIN {X 0,Y 169.258,Z 463.139,A -85,B 0,C 180,E1 -22954.765,E2 -22954.765} C_VEL
LIN {X 0,Y 170.156,Z 460.815,A -85,B 0,C 180,E1 -22959.51,E2 -22959.51} C_VEL
LIN {X 0,Y 171.314,Z 457.948,A -85,B 0,C 180,E1 -22963.041,E2 -22963.041} C_VEL
LIN {X 0,Y 173.032,Z 454.056,A -85,B 0,C 180,E1 -22966.519,E2 -22966.519} C_VEL
LIN {X 0,Y 175.271,Z 449.035,A -85,B 0,C 180,E1 -22969.928,E2 -22969.928} C_VEL
LIN {X 0,Y 178.135,Z 442.703,A -85,B 0,C 180,E1 -22973.237,E2 -22973.237} C_VEL
LIN {X 0,Y 181.455,Z 434.784,A -85,B 0,C 180,E1 -22976.45,E2 -22976.45} C_VEL
LIN {X 0,Y 184.502,Z 426.539,A -85,B 0,C 180,E1 -22979.118,E2 -22979.118} C_VEL
LIN {X 0,Y 187.891,Z 416.857,A -85,B 0,C 180,E1 -22981.579,E2 -22981.579} C_VEL
LIN {X 0,Y 187.618,Z 407.266,A -85,B 0,C 180,E1 -22984.187,E2 -22984.187} C_VEL
LIN {X 0,Y 186.363,Z 397.067,A -85,B 0,C 180,E1 -22986.74,E2 -22986.74} C_VEL
LIN {X 0,Y 184.049,Z 386.859,A -85,B 0,C 180,E1 -22989.197,E2 -22989.197} C_VEL
LIN {X 0,Y 181.053,Z 378.418,A -85,B 0,C 180,E1 -22991.292,E2 -22991.292} C_VEL
LIN {X 0,Y 176.777,Z 369.384,A -85,B 0,C 180,E1 -22993.691,E2 -22993.691} C_VEL
LIN {X 0,Y 174.713,Z 365.731,A -85,B 0,C 180,E1 -22994.745,E2 -22994.745} C_VEL
LIN {X 0,Y 173.807,Z 364.44,A -85,B 0,C 180,E1 -22995.161,E2 -22995.161} C_VEL
LIN {X 0,Y 171.987,Z 361.451,A -85,B 0,C 180,E1 -22996.058,E2 -22996.058} C_VEL
LIN {X 0,Y 171.585,Z 360.098,A -85,B 0,C 180,E1 -22996.352,E2 -22996.352} C_VEL
LIN {X 0,Y 171.343,Z 358.141,A -85,B 0,C 180,E1 -23001.199,E2 -23001.199} C_VEL
LIN {X 0,Y 171.398,Z 358.132,A -85,B 0,C 180,E1 -23005.093,E2 -23005.093} C_VEL
LIN {X 0,Y 171.409,Z 358.13,A -85,B 0,C 180,E1 -23010.527,E2 -23010.527} C_VEL
LIN {X 0,Y 171.443,Z 358.125,A -85,B 0,C 180,E1 -23015.799,E2 -23015.799} C_VEL
LIN {X 0,Y 171.579,Z 358.112,A -85,B 0,C 180,E1 -23020.871,E2 -23020.871} C_VEL
LIN {X 0,Y 171.578,Z 358.111,A -85,B 0,C 180,E1 -23025.773,E2 -23025.773} C_VEL
LIN {X 0,Y 171.889,Z 358.072,A -85,B 0,C 180,E1 -23030.587,E2 -23030.587} C_VEL
LIN {X 0,Y 171.821,Z 358.081,A -85,B 0,C 180,E1 -23035.307,E2 -23035.307} C_VEL
LIN {X 0,Y 172.325,Z 358.02,A -85,B 0,C 180,E1 -23040,E2 -23040} C_VEL
LIN {X 0,Y 171.814,Z 358.085,A -85,B 0,C 180,E1 -23044.692,E2 -23044.692} C_VEL
LIN {X 0,Y 171.848,Z 358.08,A -85,B 0,C 180,E1 -23049.415,E2 -23049.415} C_VEL
LIN {X 0,Y 171.575,Z 358.116,A -85,B 0,C 180,E1 -23054.227,E2 -23054.227} C_VEL
LIN {X 0,Y 171.542,Z 358.119,A -85,B 0,C 180,E1 -23059.558,E2 -23059.558} C_VEL
LIN {X 0,Y 171.444,Z 358.129,A -85,B 0,C 180,E1 -23065.598,E2 -23065.598} C_VEL
LIN {X 0,Y 171.39,Z 358.138,A -85,B 0,C 180,E1 -23066.812,E2 -23066.812} C_VEL
LIN {X 0,Y 171.734,Z 359.719,A -85,B 0,C 180,E1 -23070.751,E2 -23070.751} C_VEL
LIN {X 0,Y 172.058,Z 361.917,A -85,B 0,C 180,E1 -23075.221,E2 -23075.221} C_VEL
LIN {X 0,Y 172.459,Z 364.925,A -85,B 0,C 180,E1 -23080.695,E2 -23080.695} C_VEL
LIN {X 0,Y 172.855,Z 366.956,A -85,B 0,C 180,E1 -23084.129,E2 -23084.129} C_VEL
LIN {X 0,Y 174.105,Z 370.292,A -85,B 0,C 180,E1 -23084.842,E2 -23084.842} C_VEL
LIN {X 0,Y 175.815,Z 372.852,A -85,B 0,C 180,E1 -23085.618,E2 -23085.618} C_VEL
LIN {X 0,Y 177.899,Z 376.859,A -85,B 0,C 180,E1 -23086.666,E2 -23086.666} C_VEL
LIN {X 0,Y 181.452,Z 385.279,A -85,B 0,C 180,E1 -23088.669,E2 -23088.669} C_VEL
LIN {X 0,Y 183.799,Z 393.947,A -85,B 0,C 180,E1 -23090.545,E2 -23090.545} C_VEL
LIN {X 0,Y 185.399,Z 405.277,A -85,B 0,C 180,E1 -23092.929,E2 -23092.929} C_VEL
LIN {X 0,Y 185.908,Z 416.425,A -85,B 0,C 180,E1 -23095.454,E2 -23095.454} C_VEL
LIN {X 0,Y 185.499,Z 426.325,A -85,B 0,C 180,E1 -23097.966,E2 -23097.966} C_VEL
LIN {X 0,Y 184.648,Z 432.581,A -85,B 0,C 180,E1 -23099.713,E2 -23099.713} C_VEL
LIN {X 0,Y 181.328,Z 441.413,A -85,B 0,C 180,E1 -23102.283,E2 -23102.283} C_VEL
LIN {X 0,Y 178.134,Z 449.647,A -85,B 0,C 180,E1 -23105.337,E2 -23105.337} C_VEL
LIN {X 0,Y 175.029,Z 456.92,A -85,B 0,C 180,E1 -23108.814,E2 -23108.814} C_VEL
LIN {X 0,Y 172.668,Z 462.445,A -85,B 0,C 180,E1 -23112.225,E2 -23112.225} C_VEL
LIN {X 0,Y 170.947,Z 466.785,A -85,B 0,C 180,E1 -23115.719,E2 -23115.719} C_VEL
LIN {X 0,Y 170.102,Z 469.085,A -85,B 0,C 180,E1 -23118.077,E2 -23118.077} C_VEL
LIN {X 0,Y 169.488,Z 470.949,A -85,B 0,C 180,E1 -23120.452,E2 -23120.452} C_VEL
LIN {X 0,Y 169.106,Z 472.349,A -85,B 0,C 180,E1 -23122.837,E2 -23122.837} C_VEL
LIN {X 0,Y 168.892,Z 473.853,A -85,B 0,C 180,E1 -23127.078,E2 -23127.078} C_VEL
LIN {X 0,Y 168.981,Z 474.18,A -85,B 0,C 180,E1 -23129.999,E2 -23129.999} C_VEL
LIN {X 0,Y 168.892,Z 473.842,A -85,B 0,C 180,E1 -23132.92,E2 -23132.92} C_VEL
LIN {X 0,Y 169.105,Z 472.325,A -85,B 0,C 180,E1 -23137.161,E2 -23137.161} C_VEL
LIN {X 0,Y 169.486,Z 470.915,A -85,B 0,C 180,E1 -23139.546,E2 -23139.546} C_VEL
LIN {X 0,Y 170.494,Z 467.96,A -85,B 0,C 180,E1 -23143.103,E2 -23143.103} C_VEL
LIN {X 0,Y 171.967,Z 463.966,A -85,B 0,C 180,E1 -23146.622,E2 -23146.622} C_VEL
LIN {X 0,Y 173.035,Z 461.505,A -85,B 0,C 180,E1 -23148.354,E2 -23148.354} C_VEL
LIN {X 0,Y 173.556,Z 458.87,A -85,B 0,C 180,E1 -23150.099,E2 -23150.099} C_VEL
LIN {X 0,Y 172.879,Z 454.201,A -85,B 0,C 180,E1 -23152.994,E2 -23152.994} C_VEL
LIN {X 0,Y 172.44,Z 448.889,A -85,B 0,C 180,E1 -23155.781,E2 -23155.781} C_VEL
LIN {X 0,Y 173.3,Z 445.244,A -85,B 0,C 180,E1 -23157.303,E2 -23157.303} C_VEL
LIN {X 0,Y 177.047,Z 435.926,A -85,B 0,C 180,E1 -23160.404,E2 -23160.404} C_VEL
LIN {X 0,Y 178.363,Z 432.164,A -85,B 0,C 180,E1 -23161.47,E2 -23161.47} C_VEL
LIN {X 0,Y 179.332,Z 423.175,A -85,B 0,C 180,E1 -23164.049,E2 -23164.049} C_VEL
LIN {X 0,Y 179.594,Z 414.331,A -85,B 0,C 180,E1 -23166.321,E2 -23166.321} C_VEL
LIN {X 0,Y 178.927,Z 403.253,A -85,B 0,C 180,E1 -23168.934,E2 -23168.934} C_VEL
LIN {X 0,Y 177.347,Z 393.407,A -85,B 0,C 180,E1 -23171.154,E2 -23171.154} C_VEL
LIN {X 0,Y 174.952,Z 385.498,A -85,B 0,C 180,E1 -23173.069,E2 -23173.069} C_VEL
LIN {X 0,Y 172.513,Z 380.243,A -85,B 0,C 180,E1 -23174.526,E2 -23174.526} C_VEL
LIN {X 0,Y 170.675,Z 376.52,A -85,B 0,C 180,E1 -23175.571,E2 -23175.571} C_VEL
LIN {X 0,Y 168.127,Z 371.684,A -85,B 0,C 180,E1 -23176.98,E2 -23176.98} C_VEL
LIN {X 0,Y 166.093,Z 368.487,A -85,B 0,C 180,E1 -23178.043,E2 -23178.043} C_VEL
LIN {X 0,Y 165.533,Z 366.59,A -85,B 0,C 180,E1 -23178.519,E2 -23178.519} C_VEL
LIN {X 0,Y 165.131,Z 363.968,A -85,B 0,C 180,E1 -23183.427,E2 -23183.427} C_VEL
LIN {X 0,Y 164.804,Z 361.175,A -85,B 0,C 180,E1 -23189.221,E2 -23189.221} C_VEL
LIN {X 0,Y 164.389,Z 359.009,A -85,B 0,C 180,E1 -23194.69,E2 -23194.69} C_VEL
LIN {X 0,Y 164.479,Z 358.996,A -85,B 0,C 180,E1 -23200.051,E2 -23200.051} C_VEL
LIN {X 0,Y 164.53,Z 358.991,A -85,B 0,C 180,E1 -23205.15,E2 -23205.15} C_VEL
LIN {X 0,Y 164.822,Z 358.956,A -85,B 0,C 180,E1 -23210.18,E2 -23210.18} C_VEL
LIN {X 0,Y 164.846,Z 358.952,A -85,B 0,C 180,E1 -23212.652,E2 -23212.652} C_VEL
LIN {X 0,Y 165.044,Z 358.925,A -85,B 0,C 180,E1 -23217.56,E2 -23217.56} C_VEL
LIN {X 0,Y 165.283,Z 358.895,A -85,B 0,C 180,E1 -23220,E2 -23220} C_VEL
LIN {X 0,Y 164.769,Z 358.959,A -85,B 0,C 180,E1 -23224.894,E2 -23224.894} C_VEL
LIN {X 0,Y 164.855,Z 358.95,A -85,B 0,C 180,E1 -23227.348,E2 -23227.348} C_VEL
LIN {X 0,Y 164.743,Z 358.962,A -85,B 0,C 180,E1 -23231.143,E2 -23231.143} C_VEL
LIN {X 0,Y 164.478,Z 358.995,A -85,B 0,C 180,E1 -23237.404,E2 -23237.404} C_VEL
LIN {X 0,Y 164.468,Z 358.997,A -85,B 0,C 180,E1 -23239.99,E2 -23239.99} C_VEL
LIN {X 0,Y 164.365,Z 359.011,A -85,B 0,C 180,E1 -23246.118,E2 -23246.118} C_VEL
LIN {X 0,Y 164.353,Z 359.012,A -85,B 0,C 180,E1 -23251.218,E2 -23251.218} C_VEL
LIN {X 0,Y 164.276,Z 359.023,A -85,B 0,C 180,E1 -23256.795,E2 -23256.795} C_VEL
LIN {X 0,Y 164.503,Z 360.447,A -85,B 0,C 180,E1 -23261.264,E2 -23261.264} C_VEL
LIN {X 0,Y 165.697,Z 363.399,A -85,B 0,C 180,E1 -23262.018,E2 -23262.018} C_VEL
LIN {X 0,Y 167.776,Z 366.156,A -85,B 0,C 180,E1 -23263.078,E2 -23263.078} C_VEL
LIN {X 0,Y 169.753,Z 369.683,A -85,B 0,C 180,E1 -23264.203,E2 -23264.203} C_VEL
LIN {X 0,Y 173.933,Z 377.759,A -85,B 0,C 180,E1 -23266.662,E2 -23266.662} C_VEL
LIN {X 0,Y 177.13,Z 385.864,A -85,B 0,C 180,E1 -23268.927,E2 -23268.927} C_VEL
LIN {X 0,Y 179.171,Z 393.299,A -85,B 0,C 180,E1 -23270.867,E2 -23270.867} C_VEL
LIN {X 0,Y 180.769,Z 402.584,A -85,B 0,C 180,E1 -23273.285,E2 -23273.285} C_VEL
LIN {X 0,Y 181.471,Z 411.922,A -85,B 0,C 180,E1 -23275.834,E2 -23275.834} C_VEL
LIN {X 0,Y 181.465,Z 417.606,A -85,B 0,C 180,E1 -23277.497,E2 -23277.497} C_VEL
LIN {X 0,Y 177.857,Z 427.952,A -85,B 0,C 180,E1 -23280.292,E2 -23280.292} C_VEL
LIN {X 0,Y 174.68,Z 436.1,A -85,B 0,C 180,E1 -23283.089,E2 -23283.089} C_VEL
LIN {X 0,Y 171.165,Z 443.773,A -85,B 0,C 180,E1 -23286.403,E2 -23286.403} C_VEL
LIN {X 0,Y 167.834,Z 450.817,A -85,B 0,C 180,E1 -23290.429,E2 -23290.429} C_VEL
LIN {X 0,Y 165.593,Z 455.503,A -85,B 0,C 180,E1 -23293.988,E2 -23293.988} C_VEL
LIN {X 0,Y 163.925,Z 459.086,A -85,B 0,C 180,E1 -23297.623,E2 -23297.623} C_VEL
LIN {X 0,Y 163.163,Z 460.932,A -85,B 0,C 180,E1 -23300.08,E2 -23300.08} C_VEL
LIN {X 0,Y 162.612,Z 462.318,A -85,B 0,C 180,E1 -23302.551,E2 -23302.551} C_VEL
LIN {X 0,Y 161.985,Z 463.911,A -85,B 0,C 180,E1 -23307.514,E2 -23307.514} C_VEL
LIN {X 0,Y 161.964,Z 464.135,A -85,B 0,C 180,E1 -23310.001,E2 -23310.001} C_VEL
LIN {X 0,Y 162.132,Z 463.523,A -85,B 0,C 180,E1 -23314.444,E2 -23314.444} C_VEL
LIN {X 0,Y 162.556,Z 462.387,A -85,B 0,C 180,E1 -23317.453,E2 -23317.453} C_VEL
LIN {X 0,Y 163.169,Z 461.029,A -85,B 0,C 180,E1 -23319.922,E2 -23319.922} C_VEL
LIN {X 0,Y 164.41,Z 458.162,A -85,B 0,C 180,E1 -23323.599,E2 -23323.599} C_VEL
LIN {X 0,Y 166.23,Z 454.271,A -85,B 0,C 180,E1 -23327.215,E2 -23327.215} C_VEL
LIN {X 0,Y 168.607,Z 449.249,A -85,B 0,C 180,E1 -23330.751,E2 -23330.751} C_VEL
LIN {X 0,Y 171.634,Z 442.917,A -85,B 0,C 180,E1 -23334.173,E2 -23334.173} C_VEL
LIN {X 0,Y 175.125,Z 434.997,A -85,B 0,C 180,E1 -23337.485,E2 -23337.485} C_VEL
LIN {X 0,Y 178.228,Z 427.041,A -85,B 0,C 180,E1 -23340.141,E2 -23340.141} C_VEL
LIN {X 0,Y 181.51,Z 418.134,A -85,B 0,C 180,E1 -23342.496,E2 -23342.496} C_VEL
LIN {X 0,Y 181.391,Z 409.241,A -85,B 0,C 180,E1 -23345.067,E2 -23345.067} C_VEL
LIN {X 0,Y 180.389,Z 399.662,A -85,B 0,C 180,E1 -23347.642,E2 -23347.642} C_VEL
LIN {X 0,Y 178.292,Z 389.525,A -85,B 0,C 180,E1 -23350.272,E2 -23350.272} C_VEL
LIN {X 0,Y 175.784,Z 382.063,A -85,B 0,C 180,E1 -23352.3,E2 -23352.3} C_VEL
LIN {X 0,Y 172.16,Z 374.08,A -85,B 0,C 180,E1 -23354.615,E2 -23354.615} C_VEL
LIN {X 0,Y 169.611,Z 369.529,A -85,B 0,C 180,E1 -23356.068,E2 -23356.068} C_VEL
LIN {X 0,Y 167.663,Z 366.01,A -85,B 0,C 180,E1 -23357.185,E2 -23357.185} C_VEL
LIN {X 0,Y 165.139,Z 362.313,A -85,B 0,C 180,E1 -23358.523,E2 -23358.523} C_VEL
LIN {X 0,Y 164.529,Z 360.362,A -85,B 0,C 180,E1 -23359.048,E2 -23359.048} C_VEL
LIN {X 0,Y 164.28,Z 359.02,A -85,B 0,C 180,E1 -23363.206,E2 -23363.206} C_VEL
